LIN {X 7.026,Y 51.847,Z 52.000,A 180.000,B 0.000,C 180.000} C_DIS
LIN {X 6.520,Y 53.277,Z 52.000,A 180.000,B 0.000,C 180.000} C_DIS
LIN {X 6.460,Y 53.455,Z 52.000,A 180.000,B 0.000,C 180.000} C_DIS
LIN {X 5.992,Y 54.886,Z 52.000,A 180.000,B 0.000,C 180.000} C_DIS
LIN {X 5.935,Y 55.064,Z 52.000,A 180.000,B 0.000,C 180.000} C_DIS
LIN {X 5.503,Y 56.495,Z 52.000,A 180.000,B 0.000,C 180.000} C_DIS
LIN {X 5.450,Y 56.673,Z 52.000,A 180.000,B 0.000,C 180.000} C_DIS
LIN {X 5.400,Y 56.852,Z 52.000,A 180.000,B 0.000,C 180.000} C_DIS
LIN {X 5.005,Y 58.282,Z 52.000,A 180.000,B 0.000,C 180.000} C_DIS
LIN {X 4.958,Y 58.461,Z 52.000,A 180.000,B 0.000,C 180.000} C_DIS
LIN {X 4.598,Y 59.891,Z 52.000,A 180.000,B 0.000,C 180.000} C_DIS
LIN {X 4.554,Y 60.070,Z 52.000,A 180.000,B 0.000,C 180.000} C_DIS
LIN {X 4.513,Y 60.249,Z 52.000,A 180.000,B 0.000,C 180.000} C_DIS
LIN {X 4.189,Y 61.679,Z 52.000,A 180.000,B 0.000,C 180.000} C_DIS
LIN {X 4.150,Y 61.858,Z 52.000,A 180.000,B 0.000,C 180.000} C_DIS
LIN {X 3.825,Y 63.467,Z 52.000,A 180.000,B 0.000,C 180.000} C_DIS
LIN {X 3.792,Y 63.645,Z 52.000,A 180.000,B 0.000,C 180.000} C_DIS
LIN {X 3.538,Y 65.075,Z 52.000,A 180.000,B 0.000,C 180.000} C_DIS
LIN {X 3.506,Y 65.254,Z 52.000,A 180.000,B 0.000,C 180.000} C_DIS
LIN {X 3.479,Y 65.433,Z 52.000,A 180.000,B 0.000,C 180.000} C_DIS
LIN {X 3.259,Y 66.863,Z 52.000,A 180.000,B 0.000,C 180.000} C_DIS
LIN {X 3.233,Y 67.042,Z 52.000,A 180.000,B 0.000,C 180.000} C_DIS
LIN {X 3.025,Y 68.651,Z 52.000,A 180.000,B 0.000,C 180.000} C_DIS
LIN {X 3.004,Y 68.830,Z 52.000,A 180.000,B 0.000,C 180.000} C_DIS
LIN {X 2.833,Y 70.439,Z 52.000,A 180.000,B 0.000,C 180.000} C_DIS
LIN {X 2.818,Y 70.617,Z 52.000,A 180.000,B 0.000,C 180.000} C_DIS
LIN {X 2.700,Y 72.048,Z 52.000,A 180.000,B 0.000,C 180.000} C_DIS
LIN {X 2.686,Y 72.226,Z 52.000,A 180.000,B 0.000,C 180.000} C_DIS
LIN {X 2.685,Y 72.239,Z 52.000,A 180.000,B 0.000,C 180.000} C_DIS
LIN {X 2.675,Y 72.405,Z 52.000,A 180.000,B 0.000,C 180.000} C_DIS
LIN {X 2.591,Y 73.835,Z 52.000,A 180.000,B 0.000,C 180.000} C_DIS
LIN {X 2.581,Y 74.014,Z 52.000,A 180.000,B 0.000,C 180.000} C_DIS
LIN {X 2.525,Y 75.623,Z 52.000,A 180.000,B 0.000,C 180.000} C_DIS
LIN {X 2.520,Y 75.802,Z 52.000,A 180.000,B 0.000,C 180.000} C_DIS
LIN {X 2.506,Y 76.973,Z 52.000,A 180.000,B 0.000,C 180.000} C_DIS
LIN {X 2.501,Y 77.411,Z 52.000,A 180.000,B 0.000,C 180.000} C_DIS
LIN {X 2.501,Y 77.589,Z 52.000,A 180.000,B 0.000,C 180.000} C_DIS
LIN {X 2.520,Y 79.198,Z 52.000,A 180.000,B 0.000,C 180.000} C_DIS
LIN {X 2.525,Y 79.377,Z 52.000,A 180.000,B 0.000,C 180.000} C_DIS
LIN {X 2.581,Y 80.986,Z 52.000,A 180.000,B 0.000,C 180.000} C_DIS
LIN {X 2.591,Y 81.165,Z 52.000,A 180.000,B 0.000,C 180.000} C_DIS
LIN {X 2.675,Y 82.595,Z 52.000,A 180.000,B 0.000,C 180.000} C_DIS
LIN {X 2.685,Y 82.761,Z 52.000,A 180.000,B 0.000,C 180.000} C_DIS
LIN {X 2.686,Y 82.774,Z 52.000,A 180.000,B 0.000,C 180.000} C_DIS
LIN {X 2.700,Y 82.952,Z 52.000,A 180.000,B 0.000,C 180.000} C_DIS
LIN {X 2.818,Y 84.383,Z 52.000,A 180.000,B 0.000,C 180.000} C_DIS
LIN {X 2.833,Y 84.561,Z 52.000,A 180.000,B 0.000,C 180.000} C_DIS
LIN {X 3.004,Y 86.170,Z 52.000,A 180.000,B 0.000,C 180.000} C_DIS
LIN {X 3.025,Y 86.349,Z 52.000,A 180.000,B 0.000,C 180.000} C_DIS
LIN {X 3.233,Y 87.958,Z 52.000,A 180.000,B 0.000,C 180.000} C_DIS
LIN {X 3.259,Y 88.137,Z 52.000,A 180.000,B 0.000,C 180.000} C_DIS
LIN {X 3.479,Y 89.567,Z 52.000,A 180.000,B 0.000,C 180.000} C_DIS
LIN {X 3.506,Y 89.746,Z 52.000,A 180.000,B 0.000,C 180.000} C_DIS
LIN {X 3.538,Y 89.925,Z 52.000,A 180.000,B 0.000,C 180.000} C_DIS
LIN {X 3.792,Y 91.355,Z 52.000,A 180.000,B 0.000,C 180.000} C_DIS
LIN {X 3.825,Y 91.533,Z 52.000,A 180.000,B 0.000,C 180.000} C_DIS
LIN {X 4.150,Y 93.142,Z 52.000,A 180.000,B 0.000,C 180.000} C_DIS
LIN {X 4.189,Y 93.321,Z 52.000,A 180.000,B 0.000,C 180.000} C_DIS
LIN {X 4.513,Y 94.751,Z 52.000,A 180.000,B 0.000,C 180.000} C_DIS
LIN {X 4.554,Y 94.930,Z 52.000,A 180.000,B 0.000,C 180.000} C_DIS
LIN {X 4.598,Y 95.109,Z 52.000,A 180.000,B 0.000,C 180.000} C_DIS
LIN {X 4.958,Y 96.539,Z 52.000,A 180.000,B 0.000,C 180.000} C_DIS
LIN {X 5.005,Y 96.718,Z 52.000,A 180.000,B 0.000,C 180.000} C_DIS
LIN {X 5.400,Y 98.148,Z 52.000,A 180.000,B 0.000,C 180.000} C_DIS
LIN {X 5.450,Y 98.327,Z 52.000,A 180.000,B 0.000,C 180.000} C_DIS
LIN {X 5.503,Y 98.505,Z 52.000,A 180.000,B 0.000,C 180.000} C_DIS
LIN {X 5.935,Y 99.936,Z 52.000,A 180.000,B 0.000,C 180.000} C_DIS
LIN {X 5.992,Y 100.114,Z 52.000,A 180.000,B 0.000,C 180.000} C_DIS
LIN {X 6.460,Y 101.545,Z 52.000,A 180.000,B 0.000,C 180.000} C_DIS
LIN {X 6.520,Y 101.723,Z 52.000,A 180.000,B 0.000,C 180.000} C_DIS
LIN {X 7.026,Y 103.153,Z 52.000,A 180.000,B 0.000,C 180.000} C_DIS
LIN {X 7.089,Y 103.332,Z 52.000,A 180.000,B 0.000,C 180.000} C_DIS
LIN {X 7.154,Y 103.504,Z 52.000,A 180.000,B 0.000,C 180.000} C_DIS
LIN {X 7.701,Y 104.941,Z 52.000,A 180.000,B 0.000,C 180.000} C_DIS
LIN {X 7.773,Y 105.120,Z 52.000,A 180.000,B 0.000,C 180.000} C_DIS
LIN {X 8.355,Y 106.550,Z 52.000,A 180.000,B 0.000,C 180.000} C_DIS
LIN {X 8.405,Y 106.669,Z 52.000,A 180.000,B 0.000,C 180.000} C_DIS
LIN {X 9.053,Y 108.159,Z 52.000,A 180.000,B 0.000,C 180.000} C_DIS
LIN {X 9.120,Y 108.308,Z 52.000,A 180.000,B 0.000,C 180.000} C_DIS
LIN {X 9.797,Y 109.768,Z 52.000,A 180.000,B 0.000,C 180.000} C_DIS
LIN {X 9.836,Y 109.849,Z 52.000,A 180.000,B 0.000,C 180.000} C_DIS
LIN {X 10.551,Y 111.303,Z 52.000,A 180.000,B 0.000,C 180.000} C_DIS
LIN {X 10.587,Y 111.377,Z 52.000,A 180.000,B 0.000,C 180.000} C_DIS
LIN {X 10.680,Y 111.556,Z 52.000,A 180.000,B 0.000,C 180.000} C_DIS
LIN {X 11.332,Y 112.807,Z 52.000,A 180.000,B 0.000,C 180.000} C_DIS
LIN {X 11.426,Y 112.986,Z 52.000,A 180.000,B 0.000,C 180.000} C_DIS
LIN {X 12.215,Y 114.416,Z 52.000,A 180.000,B 0.000,C 180.000} C_DIS
LIN {X 12.317,Y 114.595,Z 52.000,A 180.000,B 0.000,C 180.000} C_DIS
LIN {X 13.053,Y 115.859,Z 52.000,A 180.000,B 0.000,C 180.000} C_DIS
LIN {X 13.151,Y 116.025,Z 52.000,A 180.000,B 0.000,C 180.000} C_DIS
LIN {X 13.232,Y 116.158,Z 52.000,A 180.000,B 0.000,C 180.000} C_DIS
LIN {X 14.029,Y 117.455,Z 52.000,A 180.000,B 0.000,C 180.000} C_DIS
LIN {X 14.126,Y 117.607,Z 52.000,A 180.000,B 0.000,C 180.000} C_DIS
LIN {X 14.953,Y 118.885,Z 52.000,A 180.000,B 0.000,C 180.000} C_DIS
LIN {X 15.020,Y 118.988,Z 52.000,A 180.000,B 0.000,C 180.000} C_DIS
LIN {X 15.072,Y 119.064,Z 52.000,A 180.000,B 0.000,C 180.000} C_DIS
LIN {X 15.924,Y 120.315,Z 52.000,A 180.000,B 0.000,C 180.000} C_DIS
LIN {X 16.047,Y 120.494,Z 52.000,A 180.000,B 0.000,C 180.000} C_DIS
LIN {X 16.986,Y 121.806,Z 52.000,A 180.000,B 0.000,C 180.000} C_DIS
LIN {X 17.073,Y 121.924,Z 52.000,A 180.000,B 0.000,C 180.000} C_DIS
LIN {X 18.059,Y 123.235,Z 52.000,A 180.000,B 0.000,C 180.000} C_DIS
LIN {X 18.152,Y 123.354,Z 52.000,A 180.000,B 0.000,C 180.000} C_DIS
LIN {X 19.139,Y 124.606,Z 52.000,A 180.000,B 0.000,C 180.000} C_DIS
LIN {X 19.286,Y 124.785,Z 52.000,A 180.000,B 0.000,C 180.000} C_DIS
LIN {X 20.204,Y 125.894,Z 52.000,A 180.000,B 0.000,C 180.000} C_DIS
LIN {X 20.323,Y 126.036,Z 52.000,A 180.000,B 0.000,C 180.000} C_DIS
LIN {X 21.410,Y 127.287,Z 52.000,A 180.000,B 0.000,C 180.000} C_DIS
LIN {X 21.456,Y 127.340,Z 52.000,A 180.000,B 0.000,C 180.000} C_DIS
LIN {X 21.570,Y 127.466,Z 52.000,A 180.000,B 0.000,C 180.000} C_DIS
LIN {X 22.547,Y 128.539,Z 52.000,A 180.000,B 0.000,C 180.000} C_DIS
LIN {X 22.707,Y 128.711,Z 52.000,A 180.000,B 0.000,C 180.000} C_DIS
LIN {X 23.780,Y 129.835,Z 52.000,A 180.000,B 0.000,C 180.000} C_DIS
LIN {X 23.910,Y 129.969,Z 52.000,A 180.000,B 0.000,C 180.000} C_DIS
LIN {X 25.031,Y 131.090,Z 52.000,A 180.000,B 0.000,C 180.000} C_DIS
LIN {X 25.165,Y 131.220,Z 52.000,A 180.000,B 0.000,C 180.000} C_DIS
LIN {X 26.289,Y 132.293,Z 52.000,A 180.000,B 0.000,C 180.000} C_DIS
LIN {X 26.461,Y 132.453,Z 52.000,A 180.000,B 0.000,C 180.000} C_DIS
LIN {X 27.534,Y 133.430,Z 52.000,A 180.000,B 0.000,C 180.000} C_DIS
LIN {X 27.660,Y 133.544,Z 52.000,A 180.000,B 0.000,C 180.000} C_DIS
LIN {X 27.713,Y 133.590,Z 52.000,A 180.000,B 0.000,C 180.000} C_DIS
LIN {X 28.964,Y 134.677,Z 52.000,A 180.000,B 0.000,C 180.000} C_DIS
LIN {X 29.106,Y 134.796,Z 52.000,A 180.000,B 0.000,C 180.000} C_DIS
LIN {X 30.215,Y 135.714,Z 52.000,A 180.000,B 0.000,C 180.000} C_DIS
LIN {X 30.394,Y 135.861,Z 52.000,A 180.000,B 0.000,C 180.000} C_DIS
LIN {X 31.646,Y 136.848,Z 52.000,A 180.000,B 0.000,C 180.000} C_DIS
LIN {X 31.765,Y 136.941,Z 52.000,A 180.000,B 0.000,C 180.000} C_DIS
LIN {X 33.076,Y 137.927,Z 52.000,A 180.000,B 0.000,C 180.000} C_DIS
LIN {X 33.194,Y 138.014,Z 52.000,A 180.000,B 0.000,C 180.000} C_DIS
LIN {X 34.506,Y 138.953,Z 52.000,A 180.000,B 0.000,C 180.000} C_DIS
LIN {X 34.685,Y 139.076,Z 52.000,A 180.000,B 0.000,C 180.000} C_DIS
LIN {X 35.936,Y 139.928,Z 52.000,A 180.000,B 0.000,C 180.000} C_DIS
LIN {X 36.012,Y 139.980,Z 52.000,A 180.000,B 0.000,C 180.000} C_DIS
LIN {X 36.115,Y 140.047,Z 52.000,A 180.000,B 0.000,C 180.000} C_DIS
LIN {X 37.393,Y 140.874,Z 52.000,A 180.000,B 0.000,C 180.000} C_DIS
LIN {X 37.545,Y 140.971,Z 52.000,A 180.000,B 0.000,C 180.000} C_DIS
LIN {X 38.842,Y 141.768,Z 52.000,A 180.000,B 0.000,C 180.000} C_DIS
LIN {X 38.975,Y 141.849,Z 52.000,A 180.000,B 0.000,C 180.000} C_DIS
LIN {X 39.141,Y 141.947,Z 52.000,A 180.000,B 0.000,C 180.000} C_DIS
LIN {X 40.405,Y 142.683,Z 52.000,A 180.000,B 0.000,C 180.000} C_DIS
LIN {X 40.584,Y 142.785,Z 52.000,A 180.000,B 0.000,C 180.000} C_DIS
LIN {X 42.014,Y 143.574,Z 52.000,A 180.000,B 0.000,C 180.000} C_DIS
LIN {X 42.193,Y 143.668,Z 52.000,A 180.000,B 0.000,C 180.000} C_DIS
LIN {X 43.444,Y 144.320,Z 52.000,A 180.000,B 0.000,C 180.000} C_DIS
LIN {X 43.623,Y 144.413,Z 52.000,A 180.000,B 0.000,C 180.000} C_DIS
LIN {X 43.697,Y 144.449,Z 52.000,A 180.000,B 0.000,C 180.000} C_DIS
LIN {X 45.151,Y 145.164,Z 52.000,A 180.000,B 0.000,C 180.000} C_DIS
LIN {X 45.232,Y 145.203,Z 52.000,A 180.000,B 0.000,C 180.000} C_DIS
LIN {X 46.692,Y 145.880,Z 52.000,A 180.000,B 0.000,C 180.000} C_DIS
LIN {X 46.841,Y 145.947,Z 52.000,A 180.000,B 0.000,C 180.000} C_DIS
LIN {X 48.331,Y 146.595,Z 52.000,A 180.000,B 0.000,C 180.000} C_DIS
LIN {X 48.450,Y 146.645,Z 52.000,A 180.000,B 0.000,C 180.000} C_DIS
LIN {X 49.880,Y 147.227,Z 52.000,A 180.000,B 0.000,C 180.000} C_DIS
LIN {X 50.059,Y 147.299,Z 52.000,A 180.000,B 0.000,C 180.000} C_DIS
LIN {X 51.496,Y 147.846,Z 52.000,A 180.000,B 0.000,C 180.000} C_DIS
LIN {X 51.668,Y 147.911,Z 52.000,A 180.000,B 0.000,C 180.000} C_DIS
LIN {X 51.847,Y 147.974,Z 52.000,A 180.000,B 0.000,C 180.000} C_DIS
LIN {X 53.277,Y 148.480,Z 52.000,A 180.000,B 0.000,C 180.000} C_DIS
LIN {X 53.455,Y 148.540,Z 52.000,A 180.000,B 0.000,C 180.000} C_DIS
LIN {X 54.290,Y 148.813,Z 52.000,A 180.000,B 0.000,C 180.000} C_DIS
LIN {X 54.886,Y 149.008,Z 52.000,A 180.000,B 0.000,C 180.000} C_DIS
LIN {X 55.064,Y 149.065,Z 52.000,A 180.000,B 0.000,C 180.000} C_DIS
LIN {X 56.495,Y 149.497,Z 52.000,A 180.000,B 0.000,C 180.000} C_DIS
LIN {X 56.673,Y 149.550,Z 52.000,A 180.000,B 0.000,C 180.000} C_DIS
LIN {X 56.852,Y 149.600,Z 52.000,A 180.000,B 0.000,C 180.000} C_DIS
LIN {X 58.282,Y 149.995,Z 52.000,A 180.000,B 0.000,C 180.000} C_DIS
LIN {X 58.461,Y 150.042,Z 52.000,A 180.000,B 0.000,C 180.000} C_DIS
LIN {X 59.891,Y 150.402,Z 52.000,A 180.000,B 0.000,C 180.000} C_DIS
LIN {X 60.070,Y 150.447,Z 52.000,A 180.000,B 0.000,C 180.000} C_DIS
LIN {X 60.249,Y 150.487,Z 52.000,A 180.000,B 0.000,C 180.000} C_DIS
LIN {X 61.679,Y 150.811,Z 52.000,A 180.000,B 0.000,C 180.000} C_DIS
LIN {X 61.858,Y 150.850,Z 52.000,A 180.000,B 0.000,C 180.000} C_DIS
LIN {X 63.467,Y 151.175,Z 52.000,A 180.000,B 0.000,C 180.000} C_DIS
LIN {X 63.645,Y 151.208,Z 52.000,A 180.000,B 0.000,C 180.000} C_DIS
LIN {X 65.075,Y 151.462,Z 52.000,A 180.000,B 0.000,C 180.000} C_DIS
LIN {X 65.254,Y 151.494,Z 52.000,A 180.000,B 0.000,C 180.000} C_DIS
LIN {X 65.433,Y 151.521,Z 52.000,A 180.000,B 0.000,C 180.000} C_DIS
LIN {X 66.863,Y 151.741,Z 52.000,A 180.000,B 0.000,C 180.000} C_DIS
LIN {X 67.042,Y 151.767,Z 52.000,A 180.000,B 0.000,C 180.000} C_DIS
LIN {X 68.651,Y 151.975,Z 52.000,A 180.000,B 0.000,C 180.000} C_DIS
LIN {X 68.830,Y 151.996,Z 52.000,A 180.000,B 0.000,C 180.000} C_DIS
LIN {X 70.439,Y 152.167,Z 52.000,A 180.000,B 0.000,C 180.000} C_DIS
LIN {X 70.617,Y 152.182,Z 52.000,A 180.000,B 0.000,C 180.000} C_DIS
LIN {X 72.048,Y 152.300,Z 52.000,A 180.000,B 0.000,C 180.000} C_DIS
LIN {X 72.226,Y 152.314,Z 52.000,A 180.000,B 0.000,C 180.000} C_DIS
LIN {X 72.239,Y 152.315,Z 52.000,A 180.000,B 0.000,C 180.000} C_DIS
LIN {X 72.405,Y 152.325,Z 52.000,A 180.000,B 0.000,C 180.000} C_DIS
LIN {X 73.835,Y 152.409,Z 52.000,A 180.000,B 0.000,C 180.000} C_DIS
LIN {X 74.014,Y 152.419,Z 52.000,A 180.000,B 0.000,C 180.000} C_DIS
LIN {X 75.623,Y 152.475,Z 52.000,A 180.000,B 0.000,C 180.000} C_DIS
LIN {X 75.802,Y 152.480,Z 52.000,A 180.000,B 0.000,C 180.000} C_DIS
LIN {X 77.411,Y 152.499,Z 52.000,A 180.000,B 0.000,C 180.000} C_DIS
LIN {X 77.589,Y 152.499,Z 52.000,A 180.000,B 0.000,C 180.000} C_DIS
LIN {X 79.198,Y 152.480,Z 52.000,A 180.000,B 0.000,C 180.000} C_DIS
LIN {X 79.377,Y 152.475,Z 52.000,A 180.000,B 0.000,C 180.000} C_DIS
LIN {X 80.986,Y 152.419,Z 52.000,A 180.000,B 0.000,C 180.000} C_DIS
LIN {X 81.165,Y 152.409,Z 52.000,A 180.000,B 0.000,C 180.000} C_DIS
LIN {X 82.595,Y 152.325,Z 52.000,A 180.000,B 0.000,C 180.000} C_DIS
LIN {X 82.761,Y 152.315,Z 52.000,A 180.000,B 0.000,C 180.000} C_DIS
LIN {X 82.774,Y 152.314,Z 52.000,A 180.000,B 0.000,C 180.000} C_DIS
LIN {X 82.952,Y 152.300,Z 52.000,A 180.000,B 0.000,C 180.000} C_DIS
LIN {X 84.383,Y 152.182,Z 52.000,A 180.000,B 0.000,C 180.000} C_DIS
LIN {X 84.561,Y 152.167,Z 52.000,A 180.000,B 0.000,C 180.000} C_DIS
LIN {X 86.170,Y 151.996,Z 52.000,A 180.000,B 0.000,C 180.000} C_DIS
LIN {X 86.349,Y 151.975,Z 52.000,A 180.000,B 0.000,C 180.000} C_DIS
LIN {X 87.958,Y 151.767,Z 52.000,A 180.000,B 0.000,C 180.000} C_DIS
LIN {X 88.137,Y 151.741,Z 52.000,A 180.000,B 0.000,C 180.000} C_DIS
LIN {X 89.567,Y 151.521,Z 52.000,A 180.000,B 0.000,C 180.000} C_DIS
LIN {X 89.746,Y 151.494,Z 52.000,A 180.000,B 0.000,C 180.000} C_DIS
LIN {X 89.925,Y 151.462,Z 52.000,A 180.000,B 0.000,C 180.000} C_DIS
LIN {X 91.355,Y 151.208,Z 52.000,A 180.000,B 0.000,C 180.000} C_DIS
LIN {X 91.533,Y 151.175,Z 52.000,A 180.000,B 0.000,C 180.000} C_DIS
LIN {X 93.142,Y 150.850,Z 52.000,A 180.000,B 0.000,C 180.000} C_DIS
LIN {X 93.321,Y 150.811,Z 52.000,A 180.000,B 0.000,C 180.000} C_DIS
LIN {X 94.751,Y 150.487,Z 52.000,A 180.000,B 0.000,C 180.000} C_DIS
LIN {X 94.930,Y 150.447,Z 52.000,A 180.000,B 0.000,C 180.000} C_DIS
LIN {X 95.109,Y 150.402,Z 52.000,A 180.000,B 0.000,C 180.000} C_DIS
LIN {X 96.539,Y 150.042,Z 52.000,A 180.000,B 0.000,C 180.000} C_DIS
LIN {X 96.718,Y 149.995,Z 52.000,A 180.000,B 0.000,C 180.000} C_DIS
LIN {X 98.148,Y 149.600,Z 52.000,A 180.000,B 0.000,C 180.000} C_DIS
LIN {X 98.327,Y 149.550,Z 52.000,A 180.000,B 0.000,C 180.000} C_DIS
LIN {X 98.505,Y 149.497,Z 52.000,A 180.000,B 0.000,C 180.000} C_DIS
LIN {X 99.936,Y 149.065,Z 52.000,A 180.000,B 0.000,C 180.000} C_DIS
LIN {X 100.114,Y 149.008,Z 52.000,A 180.000,B 0.000,C 180.000} C_DIS
LIN {X 101.545,Y 148.540,Z 52.000,A 180.000,B 0.000,C 180.000} C_DIS
LIN {X 101.723,Y 148.480,Z 52.000,A 180.000,B 0.000,C 180.000} C_DIS
LIN {X 103.153,Y 147.974,Z 52.000,A 180.000,B 0.000,C 180.000} C_DIS
LIN {X 103.332,Y 147.911,Z 52.000,A 180.000,B 0.000,C 180.000} C_DIS
LIN {X 103.504,Y 147.846,Z 52.000,A 180.000,B 0.000,C 180.000} C_DIS
LIN {X 104.941,Y 147.299,Z 52.000,A 180.000,B 0.000,C 180.000} C_DIS
LIN {X 105.120,Y 147.227,Z 52.000,A 180.000,B 0.000,C 180.000} C_DIS
LIN {X 106.550,Y 146.645,Z 52.000,A 180.000,B 0.000,C 180.000} C_DIS
LIN {X 106.669,Y 146.595,Z 52.000,A 180.000,B 0.000,C 180.000} C_DIS
LIN {X 108.159,Y 145.947,Z 52.000,A 180.000,B 0.000,C 180.000} C_DIS
LIN {X 108.308,Y 145.880,Z 52.000,A 180.000,B 0.000,C 180.000} C_DIS
LIN {X 109.768,Y 145.203,Z 52.000,A 180.000,B 0.000,C 180.000} C_DIS
LIN {X 109.849,Y 145.164,Z 52.000,A 180.000,B 0.000,C 180.000} C_DIS
LIN {X 111.303,Y 144.449,Z 52.000,A 180.000,B 0.000,C 180.000} C_DIS
LIN {X 111.377,Y 144.413,Z 52.000,A 180.000,B 0.000,C 180.000} C_DIS
LIN {X 111.556,Y 144.320,Z 52.000,A 180.000,B 0.000,C 180.000} C_DIS
LIN {X 112.807,Y 143.668,Z 52.000,A 180.000,B 0.000,C 180.000} C_DIS
LIN {X 112.986,Y 143.574,Z 52.000,A 180.000,B 0.000,C 180.000} C_DIS
LIN {X 114.416,Y 142.785,Z 52.000,A 180.000,B 0.000,C 180.000} C_DIS
LIN {X 114.595,Y 142.683,Z 52.000,A 180.000,B 0.000,C 180.000} C_DIS
LIN {X 115.859,Y 141.947,Z 52.000,A 180.000,B 0.000,C 180.000} C_DIS
LIN {X 116.025,Y 141.849,Z 52.000,A 180.000,B 0.000,C 180.000} C_DIS
LIN {X 116.158,Y 141.768,Z 52.000,A 180.000,B 0.000,C 180.000} C_DIS
LIN {X 117.455,Y 140.971,Z 52.000,A 180.000,B 0.000,C 180.000} C_DIS
LIN {X 117.607,Y 140.874,Z 52.000,A 180.000,B 0.000,C 180.000} C_DIS
LIN {X 118.885,Y 140.047,Z 52.000,A 180.000,B 0.000,C 180.000} C_DIS
LIN {X 118.988,Y 139.980,Z 52.000,A 180.000,B 0.000,C 180.000} C_DIS
LIN {X 119.064,Y 139.928,Z 52.000,A 180.000,B 0.000,C 180.000} C_DIS
LIN {X 120.315,Y 139.076,Z 52.000,A 180.000,B 0.000,C 180.000} C_DIS
LIN {X 120.494,Y 138.953,Z 52.000,A 180.000,B 0.000,C 180.000} C_DIS
LIN {X 121.806,Y 138.014,Z 52.000,A 180.000,B 0.000,C 180.000} C_DIS
LIN {X 121.924,Y 137.927,Z 52.000,A 180.000,B 0.000,C 180.000} C_DIS
LIN {X 123.235,Y 136.941,Z 52.000,A 180.000,B 0.000,C 180.000} C_DIS
LIN {X 123.354,Y 136.848,Z 52.000,A 180.000,B 0.000,C 180.000} C_DIS
LIN {X 124.606,Y 135.861,Z 52.000,A 180.000,B 0.000,C 180.000} C_DIS
LIN {X 124.785,Y 135.714,Z 52.000,A 180.000,B 0.000,C 180.000} C_DIS
LIN {X 125.894,Y 134.796,Z 52.000,A 180.000,B 0.000,C 180.000} C_DIS
LIN {X 126.036,Y 134.677,Z 52.000,A 180.000,B 0.000,C 180.000} C_DIS
LIN {X 127.287,Y 133.590,Z 52.000,A 180.000,B 0.000,C 180.000} C_DIS
LIN {X 127.340,Y 133.544,Z 52.000,A 180.000,B 0.000,C 180.000} C_DIS
LIN {X 127.466,Y 133.430,Z 52.000,A 180.000,B 0.000,C 180.000} C_DIS
LIN {X 128.539,Y 132.453,Z 52.000,A 180.000,B 0.000,C 180.000} C_DIS
LIN {X 128.711,Y 132.293,Z 52.000,A 180.000,B 0.000,C 180.000} C_DIS
LIN {X 129.835,Y 131.220,Z 52.000,A 180.000,B 0.000,C 180.000} C_DIS
LIN {X 129.969,Y 131.090,Z 52.000,A 180.000,B 0.000,C 180.000} C_DIS
LIN {X 131.090,Y 129.969,Z 52.000,A 180.000,B 0.000,C 180.000} C_DIS
LIN {X 131.220,Y 129.835,Z 52.000,A 180.000,B 0.000,C 180.000} C_DIS
LIN {X 132.293,Y 128.711,Z 52.000,A 180.000,B 0.000,C 180.000} C_DIS
LIN {X 132.453,Y 128.539,Z 52.000,A 180.000,B 0.000,C 180.000} C_DIS
LIN {X 133.430,Y 127.466,Z 52.000,A 180.000,B 0.000,C 180.000} C_DIS
LIN {X 133.544,Y 127.340,Z 52.000,A 180.000,B 0.000,C 180.000} C_DIS
LIN {X 133.590,Y 127.287,Z 52.000,A 180.000,B 0.000,C 180.000} C_DIS
LIN {X 134.677,Y 126.036,Z 52.000,A 180.000,B 0.000,C 180.000} C_DIS
LIN {X 134.796,Y 125.894,Z 52.000,A 180.000,B 0.000,C 180.000} C_DIS
LIN {X 135.714,Y 124.785,Z 52.000,A 180.000,B 0.000,C 180.000} C_DIS
LIN {X 135.861,Y 124.606,Z 52.000,A 180.000,B 0.000,C 180.000} C_DIS
LIN {X 136.848,Y 123.354,Z 52.000,A 180.000,B 0.000,C 180.000} C_DIS
LIN {X 136.941,Y 123.235,Z 52.000,A 180.000,B 0.000,C 180.000} C_DIS
LIN {X 137.927,Y 121.924,Z 52.000,A 180.000,B 0.000,C 180.000} C_DIS
LIN {X 138.014,Y 121.806,Z 52.000,A 180.000,B 0.000,C 180.000} C_DIS
LIN {X 138.953,Y 120.494,Z 52.000,A 180.000,B 0.000,C 180.000} C_DIS
LIN {X 139.076,Y 120.315,Z 52.000,A 180.000,B 0.000,C 180.000} C_DIS
LIN {X 139.928,Y 119.064,Z 52.000,A 180.000,B 0.000,C 180.000} C_DIS
LIN {X 139.980,Y 118.988,Z 52.000,A 180.000,B 0.000,C 180.000} C_DIS
LIN {X 140.047,Y 118.885,Z 52.000,A 180.000,B 0.000,C 180.000} C_DIS
LIN {X 140.874,Y 117.607,Z 52.000,A 180.000,B 0.000,C 180.000} C_DIS
LIN {X 140.971,Y 117.455,Z 52.000,A 180.000,B 0.000,C 180.000} C_DIS
LIN {X 141.768,Y 116.158,Z 52.000,A 180.000,B 0.000,C 180.000} C_DIS
LIN {X 141.849,Y 116.025,Z 52.000,A 180.000,B 0.000,C 180.000} C_DIS
LIN {X 141.947,Y 115.859,Z 52.000,A 180.000,B 0.000,C 180.000} C_DIS
LIN {X 142.683,Y 114.595,Z 52.000,A 180.000,B 0.000,C 180.000} C_DIS
LIN {X 142.785,Y 114.416,Z 52.000,A 180.000,B 0.000,C 180.000} C_DIS
LIN {X 143.574,Y 112.986,Z 52.000,A 180.000,B 0.000,C 180.000} C_DIS
LIN {X 143.668,Y 112.807,Z 52.000,A 180.000,B 0.000,C 180.000} C_DIS
LIN {X 144.320,Y 111.556,Z 52.000,A 180.000,B 0.000,C 180.000} C_DIS
LIN {X 144.413,Y 111.377,Z 52.000,A 180.000,B 0.000,C 180.000} C_DIS
LIN {X 144.449,Y 111.303,Z 52.000,A 180.000,B 0.000,C 180.000} C_DIS
LIN {X 145.164,Y 109.849,Z 52.000,A 180.000,B 0.000,C 180.000} C_DIS
LIN {X 145.203,Y 109.768,Z 52.000,A 180.000,B 0.000,C 180.000} C_DIS
LIN {X 145.656,Y 108.791,Z 52.000,A 180.000,B 0.000,C 180.000} C_DIS
LIN {X 145.880,Y 108.308,Z 52.000,A 180.000,B 0.000,C 180.000} C_DIS
LIN {X 145.947,Y 108.159,Z 52.000,A 180.000,B 0.000,C 180.000} C_DIS
LIN {X 146.595,Y 106.669,Z 52.000,A 180.000,B 0.000,C 180.000} C_DIS
LIN {X 146.645,Y 106.550,Z 52.000,A 180.000,B 0.000,C 180.000} C_DIS
LIN {X 147.227,Y 105.120,Z 52.000,A 180.000,B 0.000,C 180.000} C_DIS
LIN {X 147.299,Y 104.941,Z 52.000,A 180.000,B 0.000,C 180.000} C_DIS
LIN {X 147.846,Y 103.504,Z 52.000,A 180.000,B 0.000,C 180.000} C_DIS
LIN {X 147.911,Y 103.332,Z 52.000,A 180.000,B 0.000,C 180.000} C_DIS
LIN {X 147.974,Y 103.153,Z 52.000,A 180.000,B 0.000,C 180.000} C_DIS
LIN {X 148.480,Y 101.723,Z 52.000,A 180.000,B 0.000,C 180.000} C_DIS
LIN {X 148.540,Y 101.545,Z 52.000,A 180.000,B 0.000,C 180.000} C_DIS
LIN {X 149.008,Y 100.114,Z 52.000,A 180.000,B 0.000,C 180.000} C_DIS
LIN {X 149.065,Y 99.936,Z 52.000,A 180.000,B 0.000,C 180.000} C_DIS
LIN {X 149.497,Y 98.505,Z 52.000,A 180.000,B 0.000,C 180.000} C_DIS
LIN {X 149.550,Y 98.327,Z 52.000,A 180.000,B 0.000,C 180.000} C_DIS
LIN {X 149.600,Y 98.148,Z 52.000,A 180.000,B 0.000,C 180.000} C_DIS
LIN {X 149.995,Y 96.718,Z 52.000,A 180.000,B 0.000,C 180.000} C_DIS
LIN {X 150.042,Y 96.539,Z 52.000,A 180.000,B 0.000,C 180.000} C_DIS
LIN {X 150.402,Y 95.109,Z 52.000,A 180.000,B 0.000,C 180.000} C_DIS
LIN {X 150.447,Y 94.930,Z 52.000,A 180.000,B 0.000,C 180.000} C_DIS
LIN {X 150.487,Y 94.751,Z 52.000,A 180.000,B 0.000,C 180.000} C_DIS
LIN {X 150.811,Y 93.321,Z 52.000,A 180.000,B 0.000,C 180.000} C_DIS
LIN {X 150.850,Y 93.142,Z 52.000,A 180.000,B 0.000,C 180.000} C_DIS
LIN {X 151.175,Y 91.533,Z 52.000,A 180.000,B 0.000,C 180.000} C_DIS
LIN {X 151.208,Y 91.355,Z 52.000,A 180.000,B 0.000,C 180.000} C_DIS
LIN {X 151.462,Y 89.925,Z 52.000,A 180.000,B 0.000,C 180.000} C_DIS
LIN {X 151.494,Y 89.746,Z 52.000,A 180.000,B 0.000,C 180.000} C_DIS
LIN {X 151.521,Y 89.567,Z 52.000,A 180.000,B 0.000,C 180.000} C_DIS
LIN {X 151.741,Y 88.137,Z 52.000,A 180.000,B 0.000,C 180.000} C_DIS
LIN {X 151.767,Y 87.958,Z 52.000,A 180.000,B 0.000,C 180.000} C_DIS
LIN {X 151.975,Y 86.349,Z 52.000,A 180.000,B 0.000,C 180.000} C_DIS
LIN {X 151.996,Y 86.170,Z 52.000,A 180.000,B 0.000,C 180.000} C_DIS
LIN {X 152.167,Y 84.561,Z 52.000,A 180.000,B 0.000,C 180.000} C_DIS
LIN {X 152.182,Y 84.383,Z 52.000,A 180.000,B 0.000,C 180.000} C_DIS
LIN {X 152.300,Y 82.952,Z 52.000,A 180.000,B 0.000,C 180.000} C_DIS
LIN {X 152.314,Y 82.774,Z 52.000,A 180.000,B 0.000,C 180.000} C_DIS
LIN {X 152.315,Y 82.761,Z 52.000,A 180.000,B 0.000,C 180.000} C_DIS
LIN {X 152.325,Y 82.595,Z 52.000,A 180.000,B 0.000,C 180.000} C_DIS
LIN {X 152.409,Y 81.165,Z 52.000,A 180.000,B 0.000,C 180.000} C_DIS
LIN {X 152.419,Y 80.986,Z 52.000,A 180.000,B 0.000,C 180.000} C_DIS
LIN {X 152.475,Y 79.377,Z 52.000,A 180.000,B 0.000,C 180.000} C_DIS
LIN {X 152.480,Y 79.198,Z 52.000,A 180.000,B 0.000,C 180.000} C_DIS
LIN {X 152.499,Y 77.589,Z 52.000,A 180.000,B 0.000,C 180.000} C_DIS
LIN {X 152.499,Y 77.411,Z 52.000,A 180.000,B 0.000,C 180.000} C_DIS
LIN {X 152.480,Y 75.802,Z 52.000,A 180.000,B 0.000,C 180.000} C_DIS
LIN {X 152.475,Y 75.623,Z 52.000,A 180.000,B 0.000,C 180.000} C_DIS
LIN {X 152.419,Y 74.014,Z 52.000,A 180.000,B 0.000,C 180.000} C_DIS
LIN {X 152.409,Y 73.835,Z 52.000,A 180.000,B 0.000,C 180.000} C_DIS
LIN {X 152.342,Y 72.697,Z 52.000,A 180.000,B 0.000,C 180.000} C_DIS
; Lead Out Move Starts
LIN {X 152.468,Y 72.336,Z 52.000,A 180.000,B 0.000,C 180.000} C_DIS
LIN {X 152.812,Y 72.169,Z 52.000,A 180.000,B 0.000,C 180.000} C_DIS
; Link Move Starts
LIN {X 153.185,Y 71.967,Z 52.000,A 180.000,B 0.000,C 180.000} C_DIS
LIN {X 153.269,Y 71.551,Z 52.000,A 180.000,B 0.000,C 180.000} C_DIS
LIN {X 153.386,Y 71.095,Z 52.000,A 180.000,B 0.000,C 180.000} C_DIS
LIN {X 154.503,Y 70.413,Z 52.000,A 180.000,B 0.000,C 180.000} C_DIS
LIN {X 155.812,Y 70.426,Z 52.000,A 180.000,B 0.000,C 180.000} C_DIS
LIN {X 156.915,Y 71.130,Z 52.000,A 180.000,B 0.000,C 180.000} C_DIS
LIN {X 157.478,Y 72.311,Z 52.000,A 180.000,B 0.000,C 180.000} C_DIS
LIN {X 157.329,Y 73.611,Z 52.000,A 180.000,B 0.000,C 180.000} C_DIS
LIN {X 156.514,Y 74.635,Z 52.000,A 180.000,B 0.000,C 180.000} C_DIS
LIN {X 155.281,Y 75.073,Z 52.000,A 180.000,B 0.000,C 180.000} C_DIS
LIN {X 154.003,Y 74.790,Z 52.000,A 180.000,B 0.000,C 180.000} C_DIS
$VEL.CP=0.01
LIN {X 153.988,Y 74.782,Z 52.000,A 180.000,B 0.000,C 180.000} C_DIS
LIN {X 153.042,Y 73.825,Z 51.952,A 180.000,B 0.000,C 180.000} C_DIS
LIN {X 152.768,Y 72.509,Z 51.905,A 180.000,B 0.000,C 180.000} C_DIS
LIN {X 153.252,Y 71.255,Z 51.857,A 180.000,B 0.000,C 180.000} C_DIS
LIN {X 154.340,Y 70.464,Z 51.809,A 180.000,B 0.000,C 180.000} C_DIS
LIN {X 155.683,Y 70.391,Z 51.762,A 180.000,B 0.000,C 180.000} C_DIS
LIN {X 156.850,Y 71.059,Z 51.714,A 180.000,B 0.000,C 180.000} C_DIS
LIN {X 157.467,Y 72.254,Z 51.667,A 180.000,B 0.000,C 180.000} C_DIS
LIN {X 157.337,Y 73.592,Z 51.619,A 180.000,B 0.000,C 180.000} C_DIS
LIN {X 156.501,Y 74.645,Z 51.571,A 180.000,B 0.000,C 180.000} C_DIS
LIN {X 155.227,Y 75.075,Z 51.524,A 180.000,B 0.000,C 180.000} C_DIS
LIN {X 153.923,Y 74.745,Z 51.476,A 180.000,B 0.000,C 180.000} C_DIS
LIN {X 153.008,Y 73.759,Z 51.429,A 180.000,B 0.000,C 180.000} C_DIS
LIN {X 152.775,Y 72.435,Z 51.381,A 180.000,B 0.000,C 180.000} C_DIS
LIN {X 153.298,Y 71.196,Z 51.333,A 180.000,B 0.000,C 180.000} C_DIS
LIN {X 154.410,Y 70.440,Z 51.286,A 180.000,B 0.000,C 180.000} C_DIS
LIN {X 155.755,Y 70.409,Z 51.238,A 180.000,B 0.000,C 180.000} C_DIS
LIN {X 156.900,Y 71.114,Z 51.191,A 180.000,B 0.000,C 180.000} C_DIS
LIN {X 157.480,Y 72.327,Z 51.143,A 180.000,B 0.000,C 180.000} C_DIS
LIN {X 157.308,Y 73.661,Z 51.095,A 180.000,B 0.000,C 180.000} C_DIS
LIN {X 156.439,Y 74.687,Z 51.048,A 180.000,B 0.000,C 180.000} C_DIS
LIN {X 155.152,Y 75.077,Z 51.000,A 180.000,B 0.000,C 180.000} C_DIS
LIN {X 155.135,Y 75.077,Z 51.000,A 180.000,B 0.000,C 180.000} C_DIS
; Lead In Move Starts
LIN {X 154.880,Y 75.077,Z 51.000,A 180.000,B 0.000,C 180.000} C_DIS
LIN {X 153.690,Y 74.758,Z 51.000,A 180.000,B 0.000,C 180.000} C_DIS
LIN {X 152.819,Y 73.887,Z 51.000,A 180.000,B 0.000,C 180.000} C_DIS
LIN {X 152.500,Y 72.697,Z 51.000,A 180.000,B 0.000,C 180.000} C_DIS
; Cutting Move Starts
$VEL.CP=0.02
LIN {X 152.500,Y 5.009,Z 51.000,A 180.000,B 0.000,C 180.000} C_DIS
LIN {X 152.494,Y 4.830,Z 51.000,A 180.000,B 0.000,C 180.000} C_DIS
LIN {X 152.494,Y 4.827,Z 51.000,A 180.000,B 0.000,C 180.000} C_DIS
LIN {X 152.476,Y 4.651,Z 51.000,A 180.000,B 0.000,C 180.000} C_DIS
LIN {X 152.444,Y 4.472,Z 51.000,A 180.000,B 0.000,C 180.000} C_DIS
LIN {X 152.398,Y 4.294,Z 51.000,A 180.000,B 0.000,C 180.000} C_DIS
LIN {X 152.338,Y 4.115,Z 51.000,A 180.000,B 0.000,C 180.000} C_DIS
LIN {X 152.315,Y 4.057,Z 51.000,A 180.000,B 0.000,C 180.000} C_DIS
LIN {X 152.262,Y 3.936,Z 51.000,A 180.000,B 0.000,C 180.000} C_DIS
LIN {X 152.169,Y 3.757,Z 51.000,A 180.000,B 0.000,C 180.000} C_DIS
LIN {X 152.136,Y 3.702,Z 51.000,A 180.000,B 0.000,C 180.000} C_DIS
LIN {X 152.057,Y 3.579,Z 51.000,A 180.000,B 0.000,C 180.000} C_DIS
LIN {X 151.958,Y 3.445,Z 51.000,A 180.000,B 0.000,C 180.000} C_DIS
LIN {X 151.921,Y 3.400,Z 51.000,A 180.000,B 0.000,C 180.000} C_DIS
LIN {X 151.779,Y 3.243,Z 51.000,A 180.000,B 0.000,C 180.000} C_DIS
LIN {X 151.757,Y 3.221,Z 51.000,A 180.000,B 0.000,C 180.000} C_DIS
LIN {X 151.600,Y 3.079,Z 51.000,A 180.000,B 0.000,C 180.000} C_DIS
LIN {X 151.555,Y 3.042,Z 51.000,A 180.000,B 0.000,C 180.000} C_DIS
LIN {X 151.421,Y 2.943,Z 51.000,A 180.000,B 0.000,C 180.000} C_DIS
LIN {X 151.298,Y 2.864,Z 51.000,A 180.000,B 0.000,C 180.000} C_DIS
LIN {X 151.243,Y 2.831,Z 51.000,A 180.000,B 0.000,C 180.000} C_DIS
LIN {X 151.064,Y 2.738,Z 51.000,A 180.000,B 0.000,C 180.000} C_DIS
LIN {X 150.943,Y 2.685,Z 51.000,A 180.000,B 0.000,C 180.000} C_DIS
LIN {X 150.885,Y 2.662,Z 51.000,A 180.000,B 0.000,C 180.000} C_DIS
LIN {X 150.706,Y 2.602,Z 51.000,A 180.000,B 0.000,C 180.000} C_DIS
LIN {X 150.528,Y 2.556,Z 51.000,A 180.000,B 0.000,C 180.000} C_DIS
LIN {X 150.349,Y 2.524,Z 51.000,A 180.000,B 0.000,C 180.000} C_DIS
LIN {X 150.173,Y 2.506,Z 51.000,A 180.000,B 0.000,C 180.000} C_DIS
LIN {X 150.170,Y 2.506,Z 51.000,A 180.000,B 0.000,C 180.000} C_DIS
LIN {X 149.991,Y 2.500,Z 51.000,A 180.000,B 0.000,C 180.000} C_DIS
LIN {X 5.009,Y 2.500,Z 51.000,A 180.000,B 0.000,C 180.000} C_DIS
LIN {X 4.830,Y 2.506,Z 51.000,A 180.000,B 0.000,C 180.000} C_DIS
LIN {X 4.827,Y 2.506,Z 51.000,A 180.000,B 0.000,C 180.000} C_DIS
LIN {X 4.651,Y 2.524,Z 51.000,A 180.000,B 0.000,C 180.000} C_DIS
LIN {X 4.472,Y 2.556,Z 51.000,A 180.000,B 0.000,C 180.000} C_DIS
LIN {X 4.294,Y 2.602,Z 51.000,A 180.000,B 0.000,C 180.000} C_DIS
LIN {X 4.115,Y 2.662,Z 51.000,A 180.000,B 0.000,C 180.000} C_DIS
LIN {X 4.057,Y 2.685,Z 51.000,A 180.000,B 0.000,C 180.000} C_DIS
LIN {X 3.936,Y 2.738,Z 51.000,A 180.000,B 0.000,C 180.000} C_DIS
LIN {X 3.757,Y 2.831,Z 51.000,A 180.000,B 0.000,C 180.000} C_DIS
LIN {X 3.702,Y 2.864,Z 51.000,A 180.000,B 0.000,C 180.000} C_DIS
LIN {X 3.579,Y 2.943,Z 51.000,A 180.000,B 0.000,C 180.000} C_DIS
LIN {X 3.445,Y 3.042,Z 51.000,A 180.000,B 0.000,C 180.000} C_DIS
LIN {X 3.400,Y 3.079,Z 51.000,A 180.000,B 0.000,C 180.000} C_DIS
LIN {X 3.243,Y 3.221,Z 51.000,A 180.000,B 0.000,C 180.000} C_DIS
LIN {X 3.221,Y 3.243,Z 51.000,A 180.000,B 0.000,C 180.000} C_DIS
LIN {X 3.079,Y 3.400,Z 51.000,A 180.000,B 0.000,C 180.000} C_DIS
LIN {X 3.042,Y 3.445,Z 51.000,A 180.000,B 0.000,C 180.000} C_DIS
LIN {X 2.943,Y 3.579,Z 51.000,A 180.000,B 0.000,C 180.000} C_DIS
LIN {X 2.864,Y 3.702,Z 51.000,A 180.000,B 0.000,C 180.000} C_DIS
LIN {X 2.831,Y 3.757,Z 51.000,A 180.000,B 0.000,C 180.000} C_DIS
LIN {X 2.738,Y 3.936,Z 51.000,A 180.000,B 0.000,C 180.000} C_DIS
LIN {X 2.685,Y 4.057,Z 51.000,A 180.000,B 0.000,C 180.000} C_DIS
LIN {X 2.662,Y 4.115,Z 51.000,A 180.000,B 0.000,C 180.000} C_DIS
LIN {X 2.602,Y 4.294,Z 51.000,A 180.000,B 0.000,C 180.000} C_DIS
LIN {X 2.556,Y 4.472,Z 51.000,A 180.000,B 0.000,C 180.000} C_DIS
LIN {X 2.524,Y 4.651,Z 51.000,A 180.000,B 0.000,C 180.000} C_DIS
LIN {X 2.506,Y 4.827,Z 51.000,A 180.000,B 0.000,C 180.000} C_DIS
LIN {X 2.506,Y 4.830,Z 51.000,A 180.000,B 0.000,C 180.000} C_DIS
LIN {X 2.500,Y 5.009,Z 51.000,A 180.000,B 0.000,C 180.000} C_DIS
LIN {X 2.500,Y 149.991,Z 51.000,A 180.000,B 0.000,C 180.000} C_DIS
LIN {X 2.506,Y 150.170,Z 51.000,A 180.000,B 0.000,C 180.000} C_DIS
LIN {X 2.506,Y 150.173,Z 51.000,A 180.000,B 0.000,C 180.000} C_DIS
LIN {X 2.524,Y 150.349,Z 51.000,A 180.000,B 0.000,C 180.000} C_DIS
LIN {X 2.556,Y 150.528,Z 51.000,A 180.000,B 0.000,C 180.000} C_DIS
LIN {X 2.602,Y 150.706,Z 51.000,A 180.000,B 0.000,C 180.000} C_DIS
LIN {X 2.662,Y 150.885,Z 51.000,A 180.000,B 0.000,C 180.000} C_DIS
LIN {X 2.685,Y 150.943,Z 51.000,A 180.000,B 0.000,C 180.000} C_DIS
LIN {X 2.738,Y 151.064,Z 51.000,A 180.000,B 0.000,C 180.000} C_DIS
LIN {X 2.831,Y 151.243,Z 51.000,A 180.000,B 0.000,C 180.000} C_DIS
LIN {X 2.864,Y 151.298,Z 51.000,A 180.000,B 0.000,C 180.000} C_DIS
LIN {X 2.943,Y 151.421,Z 51.000,A 180.000,B 0.000,C 180.000} C_DIS
LIN {X 3.042,Y 151.555,Z 51.000,A 180.000,B 0.000,C 180.000} C_DIS
LIN {X 3.079,Y 151.600,Z 51.000,A 180.000,B 0.000,C 180.000} C_DIS
LIN {X 3.221,Y 151.757,Z 51.000,A 180.000,B 0.000,C 180.000} C_DIS
LIN {X 3.243,Y 151.779,Z 51.000,A 180.000,B 0.000,C 180.000} C_DIS
LIN {X 3.400,Y 151.921,Z 51.000,A 180.000,B 0.000,C 180.000} C_DIS
LIN {X 3.445,Y 151.958,Z 51.000,A 180.000,B 0.000,C 180.000} C_DIS
LIN {X 3.579,Y 152.057,Z 51.000,A 180.000,B 0.000,C 180.000} C_DIS
LIN {X 3.702,Y 152.136,Z 51.000,A 180.000,B 0.000,C 180.000} C_DIS
LIN {X 3.757,Y 152.169,Z 51.000,A 180.000,B 0.000,C 180.000} C_DIS
LIN {X 3.936,Y 152.262,Z 51.000,A 180.000,B 0.000,C 180.000} C_DIS
LIN {X 4.057,Y 152.315,Z 51.000,A 180.000,B 0.000,C 180.000} C_DIS
LIN {X 4.115,Y 152.338,Z 51.000,A 180.000,B 0.000,C 180.000} C_DIS
LIN {X 4.294,Y 152.398,Z 51.000,A 180.000,B 0.000,C 180.000} C_DIS
LIN {X 4.472,Y 152.444,Z 51.000,A 180.000,B 0.000,C 180.000} C_DIS
LIN {X 4.651,Y 152.476,Z 51.000,A 180.000,B 0.000,C 180.000} C_DIS
LIN {X 4.827,Y 152.494,Z 51.000,A 180.000,B 0.000,C 180.000} C_DIS
LIN {X 4.830,Y 152.494,Z 51.000,A 180.000,B 0.000,C 180.000} C_DIS
LIN {X 5.009,Y 152.500,Z 51.000,A 180.000,B 0.000,C 180.000} C_DIS
LIN {X 149.991,Y 152.500,Z 51.000,A 180.000,B 0.000,C 180.000} C_DIS
LIN {X 150.170,Y 152.494,Z 51.000,A 180.000,B 0.000,C 180.000} C_DIS
LIN {X 150.173,Y 152.494,Z 51.000,A 180.000,B 0.000,C 180.000} C_DIS
LIN {X 150.349,Y 152.476,Z 51.000,A 180.000,B 0.000,C 180.000} C_DIS
LIN {X 150.528,Y 152.444,Z 51.000,A 180.000,B 0.000,C 180.000} C_DIS
LIN {X 150.706,Y 152.398,Z 51.000,A 180.000,B 0.000,C 180.000} C_DIS
LIN {X 150.885,Y 152.338,Z 51.000,A 180.000,B 0.000,C 180.000} C_DIS
LIN {X 150.943,Y 152.315,Z 51.000,A 180.000,B 0.000,C 180.000} C_DIS
LIN {X 151.064,Y 152.262,Z 51.000,A 180.000,B 0.000,C 180.000} C_DIS
LIN {X 151.243,Y 152.169,Z 51.000,A 180.000,B 0.000,C 180.000} C_DIS
LIN {X 151.298,Y 152.136,Z 51.000,A 180.000,B 0.000,C 180.000} C_DIS
LIN {X 151.421,Y 152.057,Z 51.000,A 180.000,B 0.000,C 180.000} C_DIS
LIN {X 151.555,Y 151.958,Z 51.000,A 180.000,B 0.000,C 180.000} C_DIS
LIN {X 151.600,Y 151.921,Z 51.000,A 180.000,B 0.000,C 180.000} C_DIS
LIN {X 151.757,Y 151.779,Z 51.000,A 180.000,B 0.000,C 180.000} C_DIS
LIN {X 151.779,Y 151.757,Z 51.000,A 180.000,B 0.000,C 180.000} C_DIS
LIN {X 151.921,Y 151.600,Z 51.000,A 180.000,B 0.000,C 180.000} C_DIS
LIN {X 151.958,Y 151.555,Z 51.000,A 180.000,B 0.000,C 180.000} C_DIS
LIN {X 152.057,Y 151.421,Z 51.000,A 180.000,B 0.000,C 180.000} C_DIS
LIN {X 152.136,Y 151.298,Z 51.000,A 180.000,B 0.000,C 180.000} C_DIS
LIN {X 152.169,Y 151.243,Z 51.000,A 180.000,B 0.000,C 180.000} C_DIS
LIN {X 152.262,Y 151.064,Z 51.000,A 180.000,B 0.000,C 180.000} C_DIS
LIN {X 152.315,Y 150.943,Z 51.000,A 180.000,B 0.000,C 180.000} C_DIS
LIN {X 152.338,Y 150.885,Z 51.000,A 180.000,B 0.000,C 180.000} C_DIS
LIN {X 152.398,Y 150.706,Z 51.000,A 180.000,B 0.000,C 180.000} C_DIS
LIN {X 152.444,Y 150.528,Z 51.000,A 180.000,B 0.000,C 180.000} C_DIS
LIN {X 152.476,Y 150.349,Z 51.000,A 180.000,B 0.000,C 180.000} C_DIS
LIN {X 152.494,Y 150.173,Z 51.000,A 180.000,B 0.000,C 180.000} C_DIS
LIN {X 152.494,Y 150.170,Z 51.000,A 180.000,B 0.000,C 180.000} C_DIS
LIN {X 152.500,Y 149.991,Z 51.000,A 180.000,B 0.000,C 180.000} C_DIS
LIN {X 152.500,Y 72.697,Z 51.000,A 180.000,B 0.000,C 180.000} C_DIS
; Link Move Starts
LIN {X 152.500,Y 72.382,Z 51.000,A 180.000,B 0.000,C 180.000} C_DIS
LIN {X 152.500,Y 72.067,Z 50.999,A 180.000,B 0.000,C 180.000} C_DIS
LIN {X 152.500,Y 71.752,Z 50.998,A 180.000,B 0.000,C 180.000} C_DIS
LIN {X 152.500,Y 71.437,Z 50.996,A 180.000,B 0.000,C 180.000} C_DIS
LIN {X 152.500,Y 71.122,Z 50.994,A 180.000,B 0.000,C 180.000} C_DIS
LIN {X 152.500,Y 70.807,Z 50.991,A 180.000,B 0.000,C 180.000} C_DIS
LIN {X 152.500,Y 70.492,Z 50.988,A 180.000,B 0.000,C 180.000} C_DIS
LIN {X 152.500,Y 70.177,Z 50.985,A 180.000,B 0.000,C 180.000} C_DIS
LIN {X 152.500,Y 69.862,Z 50.981,A 180.000,B 0.000,C 180.000} C_DIS
LIN {X 152.500,Y 69.547,Z 50.977,A 180.000,B 0.000,C 180.000} C_DIS
LIN {X 152.500,Y 69.232,Z 50.972,A 180.000,B 0.000,C 180.000} C_DIS
LIN {X 152.500,Y 69.075,Z 50.969,A 180.000,B 0.000,C 180.000} C_DIS
LIN {X 152.500,Y 68.917,Z 50.967,A 180.000,B 0.000,C 180.000} C_DIS
LIN {X 152.500,Y 68.760,Z 50.964,A 180.000,B 0.000,C 180.000} C_DIS
LIN {X 152.500,Y 68.602,Z 50.961,A 180.000,B 0.000,C 180.000} C_DIS
LIN {X 152.500,Y 68.445,Z 50.959,A 180.000,B 0.000,C 180.000} C_DIS
LIN {X 152.500,Y 68.287,Z 50.956,A 180.000,B 0.000,C 180.000} C_DIS
LIN {X 152.500,Y 68.130,Z 50.952,A 180.000,B 0.000,C 180.000} C_DIS
LIN {X 152.500,Y 67.972,Z 50.949,A 180.000,B 0.000,C 180.000} C_DIS
LIN {X 152.500,Y 67.815,Z 50.946,A 180.000,B 0.000,C 180.000} C_DIS
LIN {X 152.500,Y 67.657,Z 50.943,A 180.000,B 0.000,C 180.000} C_DIS
LIN {X 152.500,Y 67.500,Z 50.939,A 180.000,B 0.000,C 180.000} C_DIS
LIN {X 152.500,Y 67.342,Z 50.936,A 180.000,B 0.000,C 180.000} C_DIS
LIN {X 152.500,Y 67.185,Z 50.932,A 180.000,B 0.000,C 180.000} C_DIS
LIN {X 152.500,Y 67.027,Z 50.928,A 180.000,B 0.000,C 180.000} C_DIS
LIN {X 152.500,Y 66.870,Z 50.925,A 180.000,B 0.000,C 180.000} C_DIS
LIN {X 152.500,Y 66.712,Z 50.921,A 180.000,B 0.000,C 180.000} C_DIS
LIN {X 152.500,Y 66.555,Z 50.917,A 180.000,B 0.000,C 180.000} C_DIS
LIN {X 152.500,Y 66.397,Z 50.913,A 180.000,B 0.000,C 180.000} C_DIS
LIN {X 152.500,Y 66.240,Z 50.909,A 180.000,B 0.000,C 180.000} C_DIS
LIN {X 152.500,Y 66.082,Z 50.905,A 180.000,B 0.000,C 180.000} C_DIS
LIN {X 152.500,Y 65.925,Z 50.900,A 180.000,B 0.000,C 180.000} C_DIS
LIN {X 152.500,Y 65.767,Z 50.896,A 180.000,B 0.000,C 180.000} C_DIS
LIN {X 152.500,Y 65.610,Z 50.892,A 180.000,B 0.000,C 180.000} C_DIS
LIN {X 152.500,Y 65.452,Z 50.887,A 180.000,B 0.000,C 180.000} C_DIS
LIN {X 152.500,Y 65.295,Z 50.883,A 180.000,B 0.000,C 180.000} C_DIS
LIN {X 152.500,Y 65.137,Z 50.878,A 180.000,B 0.000,C 180.000} C_DIS
LIN {X 152.500,Y 64.980,Z 50.873,A 180.000,B 0.000,C 180.000} C_DIS
LIN {X 152.500,Y 64.822,Z 50.869,A 180.000,B 0.000,C 180.000} C_DIS
LIN {X 152.500,Y 64.665,Z 50.864,A 180.000,B 0.000,C 180.000} C_DIS
LIN {X 152.500,Y 64.507,Z 50.859,A 180.000,B 0.000,C 180.000} C_DIS
LIN {X 152.500,Y 64.350,Z 50.854,A 180.000,B 0.000,C 180.000} C_DIS
LIN {X 152.500,Y 64.271,Z 50.851,A 180.000,B 0.000,C 180.000} C_DIS
LIN {X 152.500,Y 64.192,Z 50.849,A 180.000,B 0.000,C 180.000} C_DIS
LIN {X 152.500,Y 64.113,Z 50.846,A 180.000,B 0.000,C 180.000} C_DIS
LIN {X 152.500,Y 64.035,Z 50.844,A 180.000,B 0.000,C 180.000} C_DIS
LIN {X 152.500,Y 63.956,Z 50.841,A 180.000,B 0.000,C 180.000} C_DIS
LIN {X 152.500,Y 63.877,Z 50.839,A 180.000,B 0.000,C 180.000} C_DIS
LIN {X 152.500,Y 63.798,Z 50.836,A 180.000,B 0.000,C 180.000} C_DIS
LIN {X 152.500,Y 63.641,Z 50.831,A 180.000,B 0.000,C 180.000} C_DIS
LIN {X 152.500,Y 63.483,Z 50.825,A 180.000,B 0.000,C 180.000} C_DIS
LIN {X 152.500,Y 63.326,Z 50.820,A 180.000,B 0.000,C 180.000} C_DIS
LIN {X 152.500,Y 63.168,Z 50.815,A 180.000,B 0.000,C 180.000} C_DIS
LIN {X 152.500,Y 63.011,Z 50.809,A 180.000,B 0.000,C 180.000} C_DIS
LIN {X 152.500,Y 62.932,Z 50.806,A 180.000,B 0.000,C 180.000} C_DIS
LIN {X 152.500,Y 62.775,Z 50.801,A 180.000,B 0.000,C 180.000} C_DIS
LIN {X 152.500,Y 62.538,Z 50.793,A 180.000,B 0.000,C 180.000} C_DIS
LIN {X 152.500,Y 62.381,Z 50.787,A 180.000,B 0.000,C 180.000} C_DIS
LIN {X 152.500,Y 62.302,Z 50.785,A 180.000,B 0.000,C 180.000} C_DIS
LIN {X 152.500,Y 62.145,Z 50.779,A 180.000,B 0.000,C 180.000} C_DIS
LIN {X 152.500,Y 61.908,Z 50.771,A 180.000,B 0.000,C 180.000} C_DIS
LIN {X 152.500,Y 61.751,Z 50.765,A 180.000,B 0.000,C 180.000} C_DIS
LIN {X 152.500,Y 61.672,Z 50.763,A 180.000,B 0.000,C 180.000} C_DIS
LIN {X 152.500,Y 61.515,Z 50.757,A 180.000,B 0.000,C 180.000} C_DIS
LIN {X 152.500,Y 61.278,Z 50.749,A 180.000,B 0.000,C 180.000} C_DIS
LIN {X 152.500,Y 61.121,Z 50.743,A 180.000,B 0.000,C 180.000} C_DIS
LIN {X 152.500,Y 61.042,Z 50.741,A 180.000,B 0.000,C 180.000} C_DIS
LIN {X 152.500,Y 60.885,Z 50.735,A 180.000,B 0.000,C 180.000} C_DIS
LIN {X 152.500,Y 60.648,Z 50.727,A 180.000,B 0.000,C 180.000} C_DIS
LIN {X 152.500,Y 60.491,Z 50.721,A 180.000,B 0.000,C 180.000} C_DIS
LIN {X 152.500,Y 60.412,Z 50.719,A 180.000,B 0.000,C 180.000} C_DIS
LIN {X 152.500,Y 60.255,Z 50.713,A 180.000,B 0.000,C 180.000} C_DIS
LIN {X 152.500,Y 59.782,Z 50.697,A 180.000,B 0.000,C 180.000} C_DIS
LIN {X 152.500,Y 59.625,Z 50.691,A 180.000,B 0.000,C 180.000} C_DIS
LIN {X 152.500,Y 59.152,Z 50.675,A 180.000,B 0.000,C 180.000} C_DIS
LIN {X 152.500,Y 58.995,Z 50.669,A 180.000,B 0.000,C 180.000} C_DIS
LIN {X 152.500,Y 58.443,Z 50.650,A 180.000,B 0.000,C 180.000} C_DIS
LIN {X 152.500,Y 57.971,Z 50.633,A 180.000,B 0.000,C 180.000} C_DIS
LIN {X 152.500,Y 57.813,Z 50.628,A 180.000,B 0.000,C 180.000} C_DIS
LIN {X 152.500,Y 57.341,Z 50.611,A 180.000,B 0.000,C 180.000} C_DIS
LIN {X 152.500,Y 57.183,Z 50.606,A 180.000,B 0.000,C 180.000} C_DIS
LIN {X 152.500,Y 56.396,Z 50.578,A 180.000,B 0.000,C 180.000} C_DIS
LIN {X 152.500,Y 56.002,Z 50.565,A 180.000,B 0.000,C 180.000} C_DIS
LIN {X 152.500,Y 55.530,Z 50.548,A 180.000,B 0.000,C 180.000} C_DIS
LIN {X 152.500,Y 53.718,Z 50.485,A 180.000,B 0.000,C 180.000} C_DIS
LIN {X 152.500,Y 50.726,Z 50.380,A 180.000,B 0.000,C 180.000} C_DIS
LIN {X 152.500,Y 50.568,Z 50.375,A 180.000,B 0.000,C 180.000} C_DIS
LIN {X 152.500,Y 50.096,Z 50.358,A 180.000,B 0.000,C 180.000} C_DIS
LIN {X 152.500,Y 49.938,Z 50.353,A 180.000,B 0.000,C 180.000} C_DIS
LIN {X 152.500,Y 49.466,Z 50.336,A 180.000,B 0.000,C 180.000} C_DIS
LIN {X 152.500,Y 49.387,Z 50.334,A 180.000,B 0.000,C 180.000} C_DIS
LIN {X 152.500,Y 49.230,Z 50.328,A 180.000,B 0.000,C 180.000} C_DIS
LIN {X 152.500,Y 48.757,Z 50.312,A 180.000,B 0.000,C 180.000} C_DIS
LIN {X 152.500,Y 48.600,Z 50.306,A 180.000,B 0.000,C 180.000} C_DIS
LIN {X 152.500,Y 48.127,Z 50.290,A 180.000,B 0.000,C 180.000} C_DIS
LIN {X 152.500,Y 47.970,Z 50.284,A 180.000,B 0.000,C 180.000} C_DIS
LIN {X 152.500,Y 47.733,Z 50.276,A 180.000,B 0.000,C 180.000} C_DIS
LIN {X 152.500,Y 47.576,Z 50.270,A 180.000,B 0.000,C 180.000} C_DIS
LIN {X 152.500,Y 47.497,Z 50.268,A 180.000,B 0.000,C 180.000} C_DIS
LIN {X 152.500,Y 47.340,Z 50.262,A 180.000,B 0.000,C 180.000} C_DIS
LIN {X 152.500,Y 47.104,Z 50.254,A 180.000,B 0.000,C 180.000} C_DIS
LIN {X 152.500,Y 46.946,Z 50.248,A 180.000,B 0.000,C 180.000} C_DIS
LIN {X 152.500,Y 46.867,Z 50.246,A 180.000,B 0.000,C 180.000} C_DIS
LIN {X 152.500,Y 46.710,Z 50.240,A 180.000,B 0.000,C 180.000} C_DIS
LIN {X 152.500,Y 46.474,Z 50.232,A 180.000,B 0.000,C 180.000} C_DIS
LIN {X 152.500,Y 46.316,Z 50.226,A 180.000,B 0.000,C 180.000} C_DIS
LIN {X 152.500,Y 46.237,Z 50.224,A 180.000,B 0.000,C 180.000} C_DIS
LIN {X 152.500,Y 46.080,Z 50.218,A 180.000,B 0.000,C 180.000} C_DIS
LIN {X 152.500,Y 45.844,Z 50.210,A 180.000,B 0.000,C 180.000} C_DIS
LIN {X 152.500,Y 45.686,Z 50.204,A 180.000,B 0.000,C 180.000} C_DIS
LIN {X 152.500,Y 45.607,Z 50.202,A 180.000,B 0.000,C 180.000} C_DIS
LIN {X 152.500,Y 45.450,Z 50.196,A 180.000,B 0.000,C 180.000} C_DIS
LIN {X 152.500,Y 45.292,Z 50.191,A 180.000,B 0.000,C 180.000} C_DIS
LIN {X 152.500,Y 45.135,Z 50.185,A 180.000,B 0.000,C 180.000} C_DIS
LIN {X 152.500,Y 44.977,Z 50.180,A 180.000,B 0.000,C 180.000} C_DIS
LIN {X 152.500,Y 44.820,Z 50.174,A 180.000,B 0.000,C 180.000} C_DIS
LIN {X 152.500,Y 44.662,Z 50.169,A 180.000,B 0.000,C 180.000} C_DIS
LIN {X 152.500,Y 44.505,Z 50.164,A 180.000,B 0.000,C 180.000} C_DIS
LIN {X 152.500,Y 44.426,Z 50.161,A 180.000,B 0.000,C 180.000} C_DIS
LIN {X 152.500,Y 44.347,Z 50.159,A 180.000,B 0.000,C 180.000} C_DIS
LIN {X 152.500,Y 44.269,Z 50.156,A 180.000,B 0.000,C 180.000} C_DIS
LIN {X 152.500,Y 44.190,Z 50.154,A 180.000,B 0.000,C 180.000} C_DIS
LIN {X 152.500,Y 44.111,Z 50.151,A 180.000,B 0.000,C 180.000} C_DIS
LIN {X 152.500,Y 44.032,Z 50.148,A 180.000,B 0.000,C 180.000} C_DIS
LIN {X 152.500,Y 43.875,Z 50.143,A 180.000,B 0.000,C 180.000} C_DIS
LIN {X 152.500,Y 43.717,Z 50.139,A 180.000,B 0.000,C 180.000} C_DIS
LIN {X 152.500,Y 43.560,Z 50.134,A 180.000,B 0.000,C 180.000} C_DIS
LIN {X 152.500,Y 43.402,Z 50.129,A 180.000,B 0.000,C 180.000} C_DIS
LIN {X 152.500,Y 43.245,Z 50.124,A 180.000,B 0.000,C 180.000} C_DIS
LIN {X 152.500,Y 43.087,Z 50.120,A 180.000,B 0.000,C 180.000} C_DIS
LIN {X 152.500,Y 42.930,Z 50.115,A 180.000,B 0.000,C 180.000} C_DIS
LIN {X 152.500,Y 42.772,Z 50.110,A 180.000,B 0.000,C 180.000} C_DIS
LIN {X 152.500,Y 42.615,Z 50.106,A 180.000,B 0.000,C 180.000} C_DIS
LIN {X 152.500,Y 42.457,Z 50.102,A 180.000,B 0.000,C 180.000} C_DIS
LIN {X 152.500,Y 42.300,Z 50.097,A 180.000,B 0.000,C 180.000} C_DIS
LIN {X 152.500,Y 42.142,Z 50.093,A 180.000,B 0.000,C 180.000} C_DIS
LIN {X 152.500,Y 41.985,Z 50.089,A 180.000,B 0.000,C 180.000} C_DIS
LIN {X 152.500,Y 41.827,Z 50.085,A 180.000,B 0.000,C 180.000} C_DIS
LIN {X 152.500,Y 41.670,Z 50.081,A 180.000,B 0.000,C 180.000} C_DIS
LIN {X 152.500,Y 41.512,Z 50.077,A 180.000,B 0.000,C 180.000} C_DIS
LIN {X 152.500,Y 41.355,Z 50.073,A 180.000,B 0.000,C 180.000} C_DIS
LIN {X 152.500,Y 41.197,Z 50.070,A 180.000,B 0.000,C 180.000} C_DIS
LIN {X 152.500,Y 41.040,Z 50.066,A 180.000,B 0.000,C 180.000} C_DIS
LIN {X 152.500,Y 40.882,Z 50.062,A 180.000,B 0.000,C 180.000} C_DIS
LIN {X 152.500,Y 40.725,Z 50.059,A 180.000,B 0.000,C 180.000} C_DIS
LIN {X 152.500,Y 40.567,Z 50.056,A 180.000,B 0.000,C 180.000} C_DIS
LIN {X 152.500,Y 40.410,Z 50.052,A 180.000,B 0.000,C 180.000} C_DIS
LIN {X 152.500,Y 40.252,Z 50.049,A 180.000,B 0.000,C 180.000} C_DIS
LIN {X 152.500,Y 40.095,Z 50.046,A 180.000,B 0.000,C 180.000} C_DIS
LIN {X 152.500,Y 39.937,Z 50.043,A 180.000,B 0.000,C 180.000} C_DIS
LIN {X 152.500,Y 39.780,Z 50.040,A 180.000,B 0.000,C 180.000} C_DIS
LIN {X 152.500,Y 39.622,Z 50.037,A 180.000,B 0.000,C 180.000} C_DIS
LIN {X 152.500,Y 39.465,Z 50.034,A 180.000,B 0.000,C 180.000} C_DIS
LIN {X 152.500,Y 39.307,Z 50.032,A 180.000,B 0.000,C 180.000} C_DIS
LIN {X 152.500,Y 39.150,Z 50.029,A 180.000,B 0.000,C 180.000} C_DIS
LIN {X 152.500,Y 38.992,Z 50.027,A 180.000,B 0.000,C 180.000} C_DIS
LIN {X 152.500,Y 38.677,Z 50.022,A 180.000,B 0.000,C 180.000} C_DIS
LIN {X 152.500,Y 38.362,Z 50.018,A 180.000,B 0.000,C 180.000} C_DIS
LIN {X 152.500,Y 38.047,Z 50.014,A 180.000,B 0.000,C 180.000} C_DIS
LIN {X 152.500,Y 37.732,Z 50.011,A 180.000,B 0.000,C 180.000} C_DIS
LIN {X 152.500,Y 37.417,Z 50.008,A 180.000,B 0.000,C 180.000} C_DIS
LIN {X 152.500,Y 37.102,Z 50.005,A 180.000,B 0.000,C 180.000} C_DIS
LIN {X 152.500,Y 36.787,Z 50.003,A 180.000,B 0.000,C 180.000} C_DIS
LIN {X 152.500,Y 36.472,Z 50.002,A 180.000,B 0.000,C 180.000} C_DIS
LIN {X 152.500,Y 36.157,Z 50.001,A 180.000,B 0.000,C 180.000} C_DIS
LIN {X 152.500,Y 35.842,Z 50.000,A 180.000,B 0.000,C 180.000} C_DIS
LIN {X 152.500,Y 35.611,Z 50.000,A 180.000,B 0.000,C 180.000} C_DIS
; Cutting Move Starts
LIN {X 152.500,Y 5.009,Z 50.000,A 180.000,B 0.000,C 180.000} C_DIS
LIN {X 152.494,Y 4.830,Z 50.000,A 180.000,B 0.000,C 180.000} C_DIS
LIN {X 152.494,Y 4.827,Z 50.000,A 180.000,B 0.000,C 180.000} C_DIS
LIN {X 152.476,Y 4.651,Z 50.000,A 180.000,B 0.000,C 180.000} C_DIS
LIN {X 152.444,Y 4.472,Z 50.000,A 180.000,B 0.000,C 180.000} C_DIS
LIN {X 152.398,Y 4.294,Z 50.000,A 180.000,B 0.000,C 180.000} C_DIS
LIN {X 152.338,Y 4.115,Z 50.000,A 180.000,B 0.000,C 180.000} C_DIS
LIN {X 152.315,Y 4.057,Z 50.000,A 180.000,B 0.000,C 180.000} C_DIS
LIN {X 152.262,Y 3.936,Z 50.000,A 180.000,B 0.000,C 180.000} C_DIS
LIN {X 152.169,Y 3.757,Z 50.000,A 180.000,B 0.000,C 180.000} C_DIS
LIN {X 152.136,Y 3.702,Z 50.000,A 180.000,B 0.000,C 180.000} C_DIS
LIN {X 152.057,Y 3.579,Z 50.000,A 180.000,B 0.000,C 180.000} C_DIS
LIN {X 151.958,Y 3.445,Z 50.000,A 180.000,B 0.000,C 180.000} C_DIS
LIN {X 151.921,Y 3.400,Z 50.000,A 180.000,B 0.000,C 180.000} C_DIS
LIN {X 151.779,Y 3.243,Z 50.000,A 180.000,B 0.000,C 180.000} C_DIS
LIN {X 151.757,Y 3.221,Z 50.000,A 180.000,B 0.000,C 180.000} C_DIS
LIN {X 151.600,Y 3.079,Z 50.000,A 180.000,B 0.000,C 180.000} C_DIS
LIN {X 151.555,Y 3.042,Z 50.000,A 180.000,B 0.000,C 180.000} C_DIS
LIN {X 151.421,Y 2.943,Z 50.000,A 180.000,B 0.000,C 180.000} C_DIS
LIN {X 151.298,Y 2.864,Z 50.000,A 180.000,B 0.000,C 180.000} C_DIS
LIN {X 151.243,Y 2.831,Z 50.000,A 180.000,B 0.000,C 180.000} C_DIS
LIN {X 151.064,Y 2.738,Z 50.000,A 180.000,B 0.000,C 180.000} C_DIS
LIN {X 150.943,Y 2.685,Z 50.000,A 180.000,B 0.000,C 180.000} C_DIS
LIN {X 150.885,Y 2.662,Z 50.000,A 180.000,B 0.000,C 180.000} C_DIS
LIN {X 150.706,Y 2.602,Z 50.000,A 180.000,B 0.000,C 180.000} C_DIS
LIN {X 150.528,Y 2.556,Z 50.000,A 180.000,B 0.000,C 180.000} C_DIS
LIN {X 150.349,Y 2.524,Z 50.000,A 180.000,B 0.000,C 180.000} C_DIS
LIN {X 150.173,Y 2.506,Z 50.000,A 180.000,B 0.000,C 180.000} C_DIS
LIN {X 150.170,Y 2.506,Z 50.000,A 180.000,B 0.000,C 180.000} C_DIS
LIN {X 149.991,Y 2.500,Z 50.000,A 180.000,B 0.000,C 180.000} C_DIS
LIN {X 5.009,Y 2.500,Z 50.000,A 180.000,B 0.000,C 180.000} C_DIS
LIN {X 4.830,Y 2.506,Z 50.000,A 180.000,B 0.000,C 180.000} C_DIS
LIN {X 4.827,Y 2.506,Z 50.000,A 180.000,B 0.000,C 180.000} C_DIS
LIN {X 4.651,Y 2.524,Z 50.000,A 180.000,B 0.000,C 180.000} C_DIS
LIN {X 4.472,Y 2.556,Z 50.000,A 180.000,B 0.000,C 180.000} C_DIS
LIN {X 4.294,Y 2.602,Z 50.000,A 180.000,B 0.000,C 180.000} C_DIS
LIN {X 4.115,Y 2.662,Z 50.000,A 180.000,B 0.000,C 180.000} C_DIS
LIN {X 4.057,Y 2.685,Z 50.000,A 180.000,B 0.000,C 180.000} C_DIS
LIN {X 3.936,Y 2.738,Z 50.000,A 180.000,B 0.000,C 180.000} C_DIS
LIN {X 3.757,Y 2.831,Z 50.000,A 180.000,B 0.000,C 180.000} C_DIS
LIN {X 3.702,Y 2.864,Z 50.000,A 180.000,B 0.000,C 180.000} C_DIS
LIN {X 3.579,Y 2.943,Z 50.000,A 180.000,B 0.000,C 180.000} C_DIS
LIN {X 3.445,Y 3.042,Z 50.000,A 180.000,B 0.000,C 180.000} C_DIS
LIN {X 3.400,Y 3.079,Z 50.000,A 180.000,B 0.000,C 180.000} C_DIS
LIN {X 3.243,Y 3.221,Z 50.000,A 180.000,B 0.000,C 180.000} C_DIS
LIN {X 3.221,Y 3.243,Z 50.000,A 180.000,B 0.000,C 180.000} C_DIS
LIN {X 3.079,Y 3.400,Z 50.000,A 180.000,B 0.000,C 180.000} C_DIS
LIN {X 3.042,Y 3.445,Z 50.000,A 180.000,B 0.000,C 180.000} C_DIS
LIN {X 2.943,Y 3.579,Z 50.000,A 180.000,B 0.000,C 180.000} C_DIS
LIN {X 2.864,Y 3.702,Z 50.000,A 180.000,B 0.000,C 180.000} C_DIS
LIN {X 2.831,Y 3.757,Z 50.000,A 180.000,B 0.000,C 180.000} C_DIS
LIN {X 2.738,Y 3.936,Z 50.000,A 180.000,B 0.000,C 180.000} C_DIS
LIN {X 2.685,Y 4.057,Z 50.000,A 180.000,B 0.000,C 180.000} C_DIS
LIN {X 2.662,Y 4.115,Z 50.000,A 180.000,B 0.000,C 180.000} C_DIS
LIN {X 2.602,Y 4.294,Z 50.000,A 180.000,B 0.000,C 180.000} C_DIS
LIN {X 2.556,Y 4.472,Z 50.000,A 180.000,B 0.000,C 180.000} C_DIS
LIN {X 2.524,Y 4.651,Z 50.000,A 180.000,B 0.000,C 180.000} C_DIS
LIN {X 2.506,Y 4.827,Z 50.000,A 180.000,B 0.000,C 180.000} C_DIS
LIN {X 2.506,Y 4.830,Z 50.000,A 180.000,B 0.000,C 180.000} C_DIS
LIN {X 2.500,Y 5.009,Z 50.000,A 180.000,B 0.000,C 180.000} C_DIS
LIN {X 2.500,Y 149.991,Z 50.000,A 180.000,B 0.000,C 180.000} C_DIS
LIN {X 2.506,Y 150.170,Z 50.000,A 180.000,B 0.000,C 180.000} C_DIS
LIN {X 2.506,Y 150.173,Z 50.000,A 180.000,B 0.000,C 180.000} C_DIS
LIN {X 2.524,Y 150.349,Z 50.000,A 180.000,B 0.000,C 180.000} C_DIS
LIN {X 2.556,Y 150.528,Z 50.000,A 180.000,B 0.000,C 180.000} C_DIS
LIN {X 2.602,Y 150.706,Z 50.000,A 180.000,B 0.000,C 180.000} C_DIS
LIN {X 2.662,Y 150.885,Z 50.000,A 180.000,B 0.000,C 180.000} C_DIS
LIN {X 2.685,Y 150.943,Z 50.000,A 180.000,B 0.000,C 180.000} C_DIS
LIN {X 2.738,Y 151.064,Z 50.000,A 180.000,B 0.000,C 180.000} C_DIS
LIN {X 2.831,Y 151.243,Z 50.000,A 180.000,B 0.000,C 180.000} C_DIS
LIN {X 2.864,Y 151.298,Z 50.000,A 180.000,B 0.000,C 180.000} C_DIS
LIN {X 2.943,Y 151.421,Z 50.000,A 180.000,B 0.000,C 180.000} C_DIS
LIN {X 3.042,Y 151.555,Z 50.000,A 180.000,B 0.000,C 180.000} C_DIS
LIN {X 3.079,Y 151.600,Z 50.000,A 180.000,B 0.000,C 180.000} C_DIS
LIN {X 3.221,Y 151.757,Z 50.000,A 180.000,B 0.000,C 180.000} C_DIS
LIN {X 3.243,Y 151.779,Z 50.000,A 180.000,B 0.000,C 180.000} C_DIS
LIN {X 3.400,Y 151.921,Z 50.000,A 180.000,B 0.000,C 180.000} C_DIS
LIN {X 3.445,Y 151.958,Z 50.000,A 180.000,B 0.000,C 180.000} C_DIS
LIN {X 3.579,Y 152.057,Z 50.000,A 180.000,B 0.000,C 180.000} C_DIS
LIN {X 3.702,Y 152.136,Z 50.000,A 180.000,B 0.000,C 180.000} C_DIS
LIN {X 3.757,Y 152.169,Z 50.000,A 180.000,B 0.000,C 180.000} C_DIS
LIN {X 3.936,Y 152.262,Z 50.000,A 180.000,B 0.000,C 180.000} C_DIS
LIN {X 4.057,Y 152.315,Z 50.000,A 180.000,B 0.000,C 180.000} C_DIS
LIN {X 4.115,Y 152.338,Z 50.000,A 180.000,B 0.000,C 180.000} C_DIS
LIN {X 4.294,Y 152.398,Z 50.000,A 180.000,B 0.000,C 180.000} C_DIS
LIN {X 4.472,Y 152.444,Z 50.000,A 180.000,B 0.000,C 180.000} C_DIS
LIN {X 4.651,Y 152.476,Z 50.000,A 180.000,B 0.000,C 180.000} C_DIS
LIN {X 4.827,Y 152.494,Z 50.000,A 180.000,B 0.000,C 180.000} C_DIS
LIN {X 4.830,Y 152.494,Z 50.000,A 180.000,B 0.000,C 180.000} C_DIS
LIN {X 5.009,Y 152.500,Z 50.000,A 180.000,B 0.000,C 180.000} C_DIS
LIN {X 149.991,Y 152.500,Z 50.000,A 180.000,B 0.000,C 180.000} C_DIS
LIN {X 150.170,Y 152.494,Z 50.000,A 180.000,B 0.000,C 180.000} C_DIS
LIN {X 150.173,Y 152.494,Z 50.000,A 180.000,B 0.000,C 180.000} C_DIS
LIN {X 150.349,Y 152.476,Z 50.000,A 180.000,B 0.000,C 180.000} C_DIS
LIN {X 150.528,Y 152.444,Z 50.000,A 180.000,B 0.000,C 180.000} C_DIS
LIN {X 150.706,Y 152.398,Z 50.000,A 180.000,B 0.000,C 180.000} C_DIS
LIN {X 150.885,Y 152.338,Z 50.000,A 180.000,B 0.000,C 180.000} C_DIS
LIN {X 150.943,Y 152.315,Z 50.000,A 180.000,B 0.000,C 180.000} C_DIS
LIN {X 151.064,Y 152.262,Z 50.000,A 180.000,B 0.000,C 180.000} C_DIS
LIN {X 151.243,Y 152.169,Z 50.000,A 180.000,B 0.000,C 180.000} C_DIS
LIN {X 151.298,Y 152.136,Z 50.000,A 180.000,B 0.000,C 180.000} C_DIS
LIN {X 151.421,Y 152.057,Z 50.000,A 180.000,B 0.000,C 180.000} C_DIS
LIN {X 151.555,Y 151.958,Z 50.000,A 180.000,B 0.000,C 180.000} C_DIS
LIN {X 151.600,Y 151.921,Z 50.000,A 180.000,B 0.000,C 180.000} C_DIS
LIN {X 151.757,Y 151.779,Z 50.000,A 180.000,B 0.000,C 180.000} C_DIS
LIN {X 151.779,Y 151.757,Z 50.000,A 180.000,B 0.000,C 180.000} C_DIS
LIN {X 151.921,Y 151.600,Z 50.000,A 180.000,B 0.000,C 180.000} C_DIS
LIN {X 151.958,Y 151.555,Z 50.000,A 180.000,B 0.000,C 180.000} C_DIS
LIN {X 152.057,Y 151.421,Z 50.000,A 180.000,B 0.000,C 180.000} C_DIS
LIN {X 152.136,Y 151.298,Z 50.000,A 180.000,B 0.000,C 180.000} C_DIS
LIN {X 152.169,Y 151.243,Z 50.000,A 180.000,B 0.000,C 180.000} C_DIS
LIN {X 152.262,Y 151.064,Z 50.000,A 180.000,B 0.000,C 180.000} C_DIS
LIN {X 152.315,Y 150.943,Z 50.000,A 180.000,B 0.000,C 180.000} C_DIS
LIN {X 152.338,Y 150.885,Z 50.000,A 180.000,B 0.000,C 180.000} C_DIS
LIN {X 152.398,Y 150.706,Z 50.000,A 180.000,B 0.000,C 180.000} C_DIS
LIN {X 152.444,Y 150.528,Z 50.000,A 180.000,B 0.000,C 180.000} C_DIS
LIN {X 152.476,Y 150.349,Z 50.000,A 180.000,B 0.000,C 180.000} C_DIS
LIN {X 152.494,Y 150.173,Z 50.000,A 180.000,B 0.000,C 180.000} C_DIS
LIN {X 152.494,Y 150.170,Z 50.000,A 180.000,B 0.000,C 180.000} C_DIS
LIN {X 152.500,Y 149.991,Z 50.000,A 180.000,B 0.000,C 180.000} C_DIS
LIN {X 152.500,Y 72.697,Z 50.000,A 180.000,B 0.000,C 180.000} C_DIS
LIN {X 152.500,Y 35.611,Z 50.000,A 180.000,B 0.000,C 180.000} C_DIS
; Link Move Starts
LIN {X 152.500,Y 35.296,Z 50.000,A 180.000,B 0.000,C 180.000} C_DIS
LIN {X 152.500,Y 34.981,Z 49.999,A 180.000,B 0.000,C 180.000} C_DIS
LIN {X 152.500,Y 34.666,Z 49.998,A 180.000,B 0.000,C 180.000} C_DIS
LIN {X 152.500,Y 34.351,Z 49.996,A 180.000,B 0.000,C 180.000} C_DIS
LIN {X 152.500,Y 34.036,Z 49.994,A 180.000,B 0.000,C 180.000} C_DIS
LIN {X 152.500,Y 33.721,Z 49.991,A 180.000,B 0.000,C 180.000} C_DIS
LIN {X 152.500,Y 33.406,Z 49.988,A 180.000,B 0.000,C 180.000} C_DIS
LIN {X 152.500,Y 33.091,Z 49.985,A 180.000,B 0.000,C 180.000} C_DIS
LIN {X 152.500,Y 32.776,Z 49.981,A 180.000,B 0.000,C 180.000} C_DIS
LIN {X 152.500,Y 32.461,Z 49.977,A 180.000,B 0.000,C 180.000} C_DIS
LIN {X 152.500,Y 32.146,Z 49.972,A 180.000,B 0.000,C 180.000} C_DIS
LIN {X 152.500,Y 31.989,Z 49.969,A 180.000,B 0.000,C 180.000} C_DIS
LIN {X 152.500,Y 31.831,Z 49.967,A 180.000,B 0.000,C 180.000} C_DIS
LIN {X 152.500,Y 31.674,Z 49.964,A 180.000,B 0.000,C 180.000} C_DIS
LIN {X 152.500,Y 31.516,Z 49.961,A 180.000,B 0.000,C 180.000} C_DIS
LIN {X 152.500,Y 31.359,Z 49.959,A 180.000,B 0.000,C 180.000} C_DIS
LIN {X 152.500,Y 31.201,Z 49.956,A 180.000,B 0.000,C 180.000} C_DIS
LIN {X 152.500,Y 31.044,Z 49.952,A 180.000,B 0.000,C 180.000} C_DIS
LIN {X 152.500,Y 30.886,Z 49.949,A 180.000,B 0.000,C 180.000} C_DIS
LIN {X 152.500,Y 30.729,Z 49.946,A 180.000,B 0.000,C 180.000} C_DIS
LIN {X 152.500,Y 30.571,Z 49.943,A 180.000,B 0.000,C 180.000} C_DIS
LIN {X 152.500,Y 30.414,Z 49.939,A 180.000,B 0.000,C 180.000} C_DIS
LIN {X 152.500,Y 30.256,Z 49.936,A 180.000,B 0.000,C 180.000} C_DIS
LIN {X 152.500,Y 30.099,Z 49.932,A 180.000,B 0.000,C 180.000} C_DIS
LIN {X 152.500,Y 29.941,Z 49.928,A 180.000,B 0.000,C 180.000} C_DIS
LIN {X 152.500,Y 29.784,Z 49.925,A 180.000,B 0.000,C 180.000} C_DIS
LIN {X 152.500,Y 29.626,Z 49.921,A 180.000,B 0.000,C 180.000} C_DIS
LIN {X 152.500,Y 29.469,Z 49.917,A 180.000,B 0.000,C 180.000} C_DIS
LIN {X 152.500,Y 29.311,Z 49.913,A 180.000,B 0.000,C 180.000} C_DIS
LIN {X 152.500,Y 29.154,Z 49.909,A 180.000,B 0.000,C 180.000} C_DIS
LIN {X 152.500,Y 28.996,Z 49.905,A 180.000,B 0.000,C 180.000} C_DIS
LIN {X 152.500,Y 28.839,Z 49.900,A 180.000,B 0.000,C 180.000} C_DIS
LIN {X 152.500,Y 28.681,Z 49.896,A 180.000,B 0.000,C 180.000} C_DIS
LIN {X 152.500,Y 28.524,Z 49.892,A 180.000,B 0.000,C 180.000} C_DIS
LIN {X 152.500,Y 28.366,Z 49.887,A 180.000,B 0.000,C 180.000} C_DIS
LIN {X 152.500,Y 28.209,Z 49.883,A 180.000,B 0.000,C 180.000} C_DIS
LIN {X 152.500,Y 28.051,Z 49.878,A 180.000,B 0.000,C 180.000} C_DIS
LIN {X 152.500,Y 27.894,Z 49.873,A 180.000,B 0.000,C 180.000} C_DIS
LIN {X 152.500,Y 27.736,Z 49.869,A 180.000,B 0.000,C 180.000} C_DIS
LIN {X 152.500,Y 27.579,Z 49.864,A 180.000,B 0.000,C 180.000} C_DIS
LIN {X 152.500,Y 27.421,Z 49.859,A 180.000,B 0.000,C 180.000} C_DIS
LIN {X 152.500,Y 27.264,Z 49.854,A 180.000,B 0.000,C 180.000} C_DIS
LIN {X 152.500,Y 27.185,Z 49.851,A 180.000,B 0.000,C 180.000} C_DIS
LIN {X 152.500,Y 27.106,Z 49.849,A 180.000,B 0.000,C 180.000} C_DIS
LIN {X 152.500,Y 27.028,Z 49.846,A 180.000,B 0.000,C 180.000} C_DIS
LIN {X 152.500,Y 26.949,Z 49.844,A 180.000,B 0.000,C 180.000} C_DIS
LIN {X 152.500,Y 26.870,Z 49.841,A 180.000,B 0.000,C 180.000} C_DIS
LIN {X 152.500,Y 26.791,Z 49.839,A 180.000,B 0.000,C 180.000} C_DIS
LIN {X 152.500,Y 26.713,Z 49.836,A 180.000,B 0.000,C 180.000} C_DIS
LIN {X 152.500,Y 26.555,Z 49.831,A 180.000,B 0.000,C 180.000} C_DIS
LIN {X 152.500,Y 26.398,Z 49.825,A 180.000,B 0.000,C 180.000} C_DIS
LIN {X 152.500,Y 26.240,Z 49.820,A 180.000,B 0.000,C 180.000} C_DIS
LIN {X 152.500,Y 26.083,Z 49.815,A 180.000,B 0.000,C 180.000} C_DIS
LIN {X 152.500,Y 25.925,Z 49.809,A 180.000,B 0.000,C 180.000} C_DIS
LIN {X 152.500,Y 25.846,Z 49.806,A 180.000,B 0.000,C 180.000} C_DIS
LIN {X 152.500,Y 25.689,Z 49.801,A 180.000,B 0.000,C 180.000} C_DIS
LIN {X 152.500,Y 25.453,Z 49.793,A 180.000,B 0.000,C 180.000} C_DIS
LIN {X 152.500,Y 25.295,Z 49.787,A 180.000,B 0.000,C 180.000} C_DIS
LIN {X 152.500,Y 25.216,Z 49.785,A 180.000,B 0.000,C 180.000} C_DIS
LIN {X 152.500,Y 25.059,Z 49.779,A 180.000,B 0.000,C 180.000} C_DIS
LIN {X 152.500,Y 24.823,Z 49.771,A 180.000,B 0.000,C 180.000} C_DIS
LIN {X 152.500,Y 24.665,Z 49.765,A 180.000,B 0.000,C 180.000} C_DIS
LIN {X 152.500,Y 24.586,Z 49.763,A 180.000,B 0.000,C 180.000} C_DIS
LIN {X 152.500,Y 24.429,Z 49.757,A 180.000,B 0.000,C 180.000} C_DIS
LIN {X 152.500,Y 24.193,Z 49.749,A 180.000,B 0.000,C 180.000} C_DIS
LIN {X 152.500,Y 24.035,Z 49.743,A 180.000,B 0.000,C 180.000} C_DIS
LIN {X 152.500,Y 23.956,Z 49.741,A 180.000,B 0.000,C 180.000} C_DIS
LIN {X 152.500,Y 23.799,Z 49.735,A 180.000,B 0.000,C 180.000} C_DIS
LIN {X 152.500,Y 23.563,Z 49.727,A 180.000,B 0.000,C 180.000} C_DIS
LIN {X 152.500,Y 23.405,Z 49.721,A 180.000,B 0.000,C 180.000} C_DIS
LIN {X 152.500,Y 23.326,Z 49.719,A 180.000,B 0.000,C 180.000} C_DIS
LIN {X 152.500,Y 23.169,Z 49.713,A 180.000,B 0.000,C 180.000} C_DIS
LIN {X 152.500,Y 22.696,Z 49.697,A 180.000,B 0.000,C 180.000} C_DIS
LIN {X 152.500,Y 22.539,Z 49.691,A 180.000,B 0.000,C 180.000} C_DIS
LIN {X 152.500,Y 22.066,Z 49.675,A 180.000,B 0.000,C 180.000} C_DIS
LIN {X 152.500,Y 21.909,Z 49.669,A 180.000,B 0.000,C 180.000} C_DIS
LIN {X 152.500,Y 21.358,Z 49.650,A 180.000,B 0.000,C 180.000} C_DIS
LIN {X 152.500,Y 20.885,Z 49.633,A 180.000,B 0.000,C 180.000} C_DIS
LIN {X 152.500,Y 20.728,Z 49.628,A 180.000,B 0.000,C 180.000} C_DIS
LIN {X 152.500,Y 20.255,Z 49.611,A 180.000,B 0.000,C 180.000} C_DIS
LIN {X 152.500,Y 20.098,Z 49.606,A 180.000,B 0.000,C 180.000} C_DIS
LIN {X 152.500,Y 19.310,Z 49.578,A 180.000,B 0.000,C 180.000} C_DIS
LIN {X 152.500,Y 18.916,Z 49.565,A 180.000,B 0.000,C 180.000} C_DIS
LIN {X 152.500,Y 18.444,Z 49.548,A 180.000,B 0.000,C 180.000} C_DIS
LIN {X 152.500,Y 16.633,Z 49.485,A 180.000,B 0.000,C 180.000} C_DIS
LIN {X 152.500,Y 13.640,Z 49.380,A 180.000,B 0.000,C 180.000} C_DIS
LIN {X 152.500,Y 13.483,Z 49.375,A 180.000,B 0.000,C 180.000} C_DIS
LIN {X 152.500,Y 13.010,Z 49.358,A 180.000,B 0.000,C 180.000} C_DIS
LIN {X 152.500,Y 12.853,Z 49.353,A 180.000,B 0.000,C 180.000} C_DIS
LIN {X 152.500,Y 12.380,Z 49.336,A 180.000,B 0.000,C 180.000} C_DIS
LIN {X 152.500,Y 12.302,Z 49.334,A 180.000,B 0.000,C 180.000} C_DIS
LIN {X 152.500,Y 12.144,Z 49.328,A 180.000,B 0.000,C 180.000} C_DIS
LIN {X 152.500,Y 11.672,Z 49.312,A 180.000,B 0.000,C 180.000} C_DIS
LIN {X 152.500,Y 11.514,Z 49.306,A 180.000,B 0.000,C 180.000} C_DIS
LIN {X 152.500,Y 11.042,Z 49.290,A 180.000,B 0.000,C 180.000} C_DIS
LIN {X 152.500,Y 10.884,Z 49.284,A 180.000,B 0.000,C 180.000} C_DIS
LIN {X 152.500,Y 10.648,Z 49.276,A 180.000,B 0.000,C 180.000} C_DIS
LIN {X 152.500,Y 10.490,Z 49.270,A 180.000,B 0.000,C 180.000} C_DIS
LIN {X 152.500,Y 10.412,Z 49.268,A 180.000,B 0.000,C 180.000} C_DIS
LIN {X 152.500,Y 10.254,Z 49.262,A 180.000,B 0.000,C 180.000} C_DIS
LIN {X 152.500,Y 10.018,Z 49.254,A 180.000,B 0.000,C 180.000} C_DIS
LIN {X 152.500,Y 9.860,Z 49.248,A 180.000,B 0.000,C 180.000} C_DIS
LIN {X 152.500,Y 9.782,Z 49.246,A 180.000,B 0.000,C 180.000} C_DIS
LIN {X 152.500,Y 9.624,Z 49.240,A 180.000,B 0.000,C 180.000} C_DIS
LIN {X 152.500,Y 9.388,Z 49.232,A 180.000,B 0.000,C 180.000} C_DIS
LIN {X 152.500,Y 9.230,Z 49.226,A 180.000,B 0.000,C 180.000} C_DIS
LIN {X 152.500,Y 9.152,Z 49.224,A 180.000,B 0.000,C 180.000} C_DIS
LIN {X 152.500,Y 8.994,Z 49.218,A 180.000,B 0.000,C 180.000} C_DIS
LIN {X 152.500,Y 8.758,Z 49.210,A 180.000,B 0.000,C 180.000} C_DIS
LIN {X 152.500,Y 8.600,Z 49.204,A 180.000,B 0.000,C 180.000} C_DIS
LIN {X 152.500,Y 8.522,Z 49.202,A 180.000,B 0.000,C 180.000} C_DIS
LIN {X 152.500,Y 8.364,Z 49.196,A 180.000,B 0.000,C 180.000} C_DIS
LIN {X 152.500,Y 8.207,Z 49.191,A 180.000,B 0.000,C 180.000} C_DIS
LIN {X 152.500,Y 8.049,Z 49.185,A 180.000,B 0.000,C 180.000} C_DIS
LIN {X 152.500,Y 7.892,Z 49.180,A 180.000,B 0.000,C 180.000} C_DIS
LIN {X 152.500,Y 7.734,Z 49.174,A 180.000,B 0.000,C 180.000} C_DIS
LIN {X 152.500,Y 7.577,Z 49.169,A 180.000,B 0.000,C 180.000} C_DIS
LIN {X 152.500,Y 7.419,Z 49.164,A 180.000,B 0.000,C 180.000} C_DIS
LIN {X 152.500,Y 7.340,Z 49.161,A 180.000,B 0.000,C 180.000} C_DIS
LIN {X 152.500,Y 7.262,Z 49.159,A 180.000,B 0.000,C 180.000} C_DIS
LIN {X 152.500,Y 7.183,Z 49.156,A 180.000,B 0.000,C 180.000} C_DIS
LIN {X 152.500,Y 7.104,Z 49.154,A 180.000,B 0.000,C 180.000} C_DIS
LIN {X 152.500,Y 7.025,Z 49.151,A 180.000,B 0.000,C 180.000} C_DIS
LIN {X 152.500,Y 6.947,Z 49.148,A 180.000,B 0.000,C 180.000} C_DIS
LIN {X 152.500,Y 6.789,Z 49.143,A 180.000,B 0.000,C 180.000} C_DIS
LIN {X 152.500,Y 6.632,Z 49.139,A 180.000,B 0.000,C 180.000} C_DIS
LIN {X 152.500,Y 6.474,Z 49.134,A 180.000,B 0.000,C 180.000} C_DIS
LIN {X 152.500,Y 6.317,Z 49.129,A 180.000,B 0.000,C 180.000} C_DIS
LIN {X 152.500,Y 6.159,Z 49.124,A 180.000,B 0.000,C 180.000} C_DIS
LIN {X 152.500,Y 6.002,Z 49.120,A 180.000,B 0.000,C 180.000} C_DIS
LIN {X 152.500,Y 5.844,Z 49.115,A 180.000,B 0.000,C 180.000} C_DIS
LIN {X 152.500,Y 5.687,Z 49.110,A 180.000,B 0.000,C 180.000} C_DIS
LIN {X 152.500,Y 5.529,Z 49.106,A 180.000,B 0.000,C 180.000} C_DIS
LIN {X 152.500,Y 5.372,Z 49.102,A 180.000,B 0.000,C 180.000} C_DIS
LIN {X 152.500,Y 5.214,Z 49.097,A 180.000,B 0.000,C 180.000} C_DIS
LIN {X 152.500,Y 5.057,Z 49.093,A 180.000,B 0.000,C 180.000} C_DIS
LIN {X 152.498,Y 4.899,Z 49.089,A 180.000,B 0.000,C 180.000} C_DIS
LIN {X 152.487,Y 4.742,Z 49.085,A 180.000,B 0.000,C 180.000} C_DIS
LIN {X 152.465,Y 4.586,Z 49.081,A 180.000,B 0.000,C 180.000} C_DIS
LIN {X 152.434,Y 4.431,Z 49.077,A 180.000,B 0.000,C 180.000} C_DIS
LIN {X 152.394,Y 4.279,Z 49.073,A 180.000,B 0.000,C 180.000} C_DIS
LIN {X 152.344,Y 4.130,Z 49.070,A 180.000,B 0.000,C 180.000} C_DIS
LIN {X 152.284,Y 3.984,Z 49.066,A 180.000,B 0.000,C 180.000} C_DIS
LIN {X 152.216,Y 3.842,Z 49.062,A 180.000,B 0.000,C 180.000} C_DIS
LIN {X 152.138,Y 3.705,Z 49.059,A 180.000,B 0.000,C 180.000} C_DIS
LIN {X 152.053,Y 3.573,Z 49.056,A 180.000,B 0.000,C 180.000} C_DIS
LIN {X 151.959,Y 3.447,Z 49.052,A 180.000,B 0.000,C 180.000} C_DIS
LIN {X 151.857,Y 3.326,Z 49.049,A 180.000,B 0.000,C 180.000} C_DIS
LIN {X 151.748,Y 3.213,Z 49.046,A 180.000,B 0.000,C 180.000} C_DIS
LIN {X 151.632,Y 3.106,Z 49.043,A 180.000,B 0.000,C 180.000} C_DIS
LIN {X 151.509,Y 3.007,Z 49.040,A 180.000,B 0.000,C 180.000} C_DIS
LIN {X 151.381,Y 2.916,Z 49.037,A 180.000,B 0.000,C 180.000} C_DIS
LIN {X 151.247,Y 2.833,Z 49.034,A 180.000,B 0.000,C 180.000} C_DIS
LIN {X 151.108,Y 2.759,Z 49.032,A 180.000,B 0.000,C 180.000} C_DIS
LIN {X 150.965,Y 2.694,Z 49.029,A 180.000,B 0.000,C 180.000} C_DIS
LIN {X 150.818,Y 2.637,Z 49.027,A 180.000,B 0.000,C 180.000} C_DIS
LIN {X 150.667,Y 2.591,Z 49.024,A 180.000,B 0.000,C 180.000} C_DIS
LIN {X 150.514,Y 2.553,Z 49.022,A 180.000,B 0.000,C 180.000} C_DIS
LIN {X 150.359,Y 2.526,Z 49.020,A 180.000,B 0.000,C 180.000} C_DIS
LIN {X 150.203,Y 2.508,Z 49.018,A 180.000,B 0.000,C 180.000} C_DIS
LIN {X 149.888,Y 2.500,Z 49.014,A 180.000,B 0.000,C 180.000} C_DIS
LIN {X 149.573,Y 2.500,Z 49.011,A 180.000,B 0.000,C 180.000} C_DIS
LIN {X 149.258,Y 2.500,Z 49.008,A 180.000,B 0.000,C 180.000} C_DIS
LIN {X 148.943,Y 2.500,Z 49.005,A 180.000,B 0.000,C 180.000} C_DIS
LIN {X 148.628,Y 2.500,Z 49.003,A 180.000,B 0.000,C 180.000} C_DIS
LIN {X 148.313,Y 2.500,Z 49.002,A 180.000,B 0.000,C 180.000} C_DIS
LIN {X 147.998,Y 2.500,Z 49.001,A 180.000,B 0.000,C 180.000} C_DIS
LIN {X 147.683,Y 2.500,Z 49.000,A 180.000,B 0.000,C 180.000} C_DIS
LIN {X 147.452,Y 2.500,Z 49.000,A 180.000,B 0.000,C 180.000} C_DIS
; Cutting Move Starts
LIN {X 5.009,Y 2.500,Z 49.000,A 180.000,B 0.000,C 180.000} C_DIS
LIN {X 4.830,Y 2.506,Z 49.000,A 180.000,B 0.000,C 180.000} C_DIS
LIN {X 4.827,Y 2.506,Z 49.000,A 180.000,B 0.000,C 180.000} C_DIS
LIN {X 4.651,Y 2.524,Z 49.000,A 180.000,B 0.000,C 180.000} C_DIS
LIN {X 4.472,Y 2.556,Z 49.000,A 180.000,B 0.000,C 180.000} C_DIS
LIN {X 4.294,Y 2.602,Z 49.000,A 180.000,B 0.000,C 180.000} C_DIS
LIN {X 4.115,Y 2.662,Z 49.000,A 180.000,B 0.000,C 180.000} C_DIS
LIN {X 4.057,Y 2.685,Z 49.000,A 180.000,B 0.000,C 180.000} C_DIS
LIN {X 3.936,Y 2.738,Z 49.000,A 180.000,B 0.000,C 180.000} C_DIS
LIN {X 3.757,Y 2.831,Z 49.000,A 180.000,B 0.000,C 180.000} C_DIS
LIN {X 3.702,Y 2.864,Z 49.000,A 180.000,B 0.000,C 180.000} C_DIS
LIN {X 3.579,Y 2.943,Z 49.000,A 180.000,B 0.000,C 180.000} C_DIS
LIN {X 3.445,Y 3.042,Z 49.000,A 180.000,B 0.000,C 180.000} C_DIS
LIN {X 3.400,Y 3.079,Z 49.000,A 180.000,B 0.000,C 180.000} C_DIS
LIN {X 3.243,Y 3.221,Z 49.000,A 180.000,B 0.000,C 180.000} C_DIS
LIN {X 3.221,Y 3.243,Z 49.000,A 180.000,B 0.000,C 180.000} C_DIS
LIN {X 3.079,Y 3.400,Z 49.000,A 180.000,B 0.000,C 180.000} C_DIS
LIN {X 3.042,Y 3.445,Z 49.000,A 180.000,B 0.000,C 180.000} C_DIS
LIN {X 2.943,Y 3.579,Z 49.000,A 180.000,B 0.000,C 180.000} C_DIS
LIN {X 2.864,Y 3.702,Z 49.000,A 180.000,B 0.000,C 180.000} C_DIS
LIN {X 2.831,Y 3.757,Z 49.000,A 180.000,B 0.000,C 180.000} C_DIS
LIN {X 2.738,Y 3.936,Z 49.000,A 180.000,B 0.000,C 180.000} C_DIS
LIN {X 2.685,Y 4.057,Z 49.000,A 180.000,B 0.000,C 180.000} C_DIS
LIN {X 2.662,Y 4.115,Z 49.000,A 180.000,B 0.000,C 180.000} C_DIS
LIN {X 2.602,Y 4.294,Z 49.000,A 180.000,B 0.000,C 180.000} C_DIS
LIN {X 2.556,Y 4.472,Z 49.000,A 180.000,B 0.000,C 180.000} C_DIS
LIN {X 2.524,Y 4.651,Z 49.000,A 180.000,B 0.000,C 180.000} C_DIS
LIN {X 2.506,Y 4.827,Z 49.000,A 180.000,B 0.000,C 180.000} C_DIS
LIN {X 2.506,Y 4.830,Z 49.000,A 180.000,B 0.000,C 180.000} C_DIS
LIN {X 2.500,Y 5.009,Z 49.000,A 180.000,B 0.000,C 180.000} C_DIS
LIN {X 2.500,Y 149.991,Z 49.000,A 180.000,B 0.000,C 180.000} C_DIS
LIN {X 2.506,Y 150.170,Z 49.000,A 180.000,B 0.000,C 180.000} C_DIS
LIN {X 2.506,Y 150.173,Z 49.000,A 180.000,B 0.000,C 180.000} C_DIS
LIN {X 2.524,Y 150.349,Z 49.000,A 180.000,B 0.000,C 180.000} C_DIS
LIN {X 2.556,Y 150.528,Z 49.000,A 180.000,B 0.000,C 180.000} C_DIS
LIN {X 2.602,Y 150.706,Z 49.000,A 180.000,B 0.000,C 180.000} C_DIS
LIN {X 2.662,Y 150.885,Z 49.000,A 180.000,B 0.000,C 180.000} C_DIS
LIN {X 2.685,Y 150.943,Z 49.000,A 180.000,B 0.000,C 180.000} C_DIS
LIN {X 2.738,Y 151.064,Z 49.000,A 180.000,B 0.000,C 180.000} C_DIS
LIN {X 2.831,Y 151.243,Z 49.000,A 180.000,B 0.000,C 180.000} C_DIS
LIN {X 2.864,Y 151.298,Z 49.000,A 180.000,B 0.000,C 180.000} C_DIS
LIN {X 2.943,Y 151.421,Z 49.000,A 180.000,B 0.000,C 180.000} C_DIS
LIN {X 3.042,Y 151.555,Z 49.000,A 180.000,B 0.000,C 180.000} C_DIS
LIN {X 3.079,Y 151.600,Z 49.000,A 180.000,B 0.000,C 180.000} C_DIS
LIN {X 3.221,Y 151.757,Z 49.000,A 180.000,B 0.000,C 180.000} C_DIS
LIN {X 3.243,Y 151.779,Z 49.000,A 180.000,B 0.000,C 180.000} C_DIS
LIN {X 3.400,Y 151.921,Z 49.000,A 180.000,B 0.000,C 180.000} C_DIS
LIN {X 3.445,Y 151.958,Z 49.000,A 180.000,B 0.000,C 180.000} C_DIS
LIN {X 3.579,Y 152.057,Z 49.000,A 180.000,B 0.000,C 180.000} C_DIS
LIN {X 3.702,Y 152.136,Z 49.000,A 180.000,B 0.000,C 180.000} C_DIS
LIN {X 3.757,Y 152.169,Z 49.000,A 180.000,B 0.000,C 180.000} C_DIS
LIN {X 3.936,Y 152.262,Z 49.000,A 180.000,B 0.000,C 180.000} C_DIS
LIN {X 4.057,Y 152.315,Z 49.000,A 180.000,B 0.000,C 180.000} C_DIS
LIN {X 4.115,Y 152.338,Z 49.000,A 180.000,B 0.000,C 180.000} C_DIS
LIN {X 4.294,Y 152.398,Z 49.000,A 180.000,B 0.000,C 180.000} C_DIS
LIN {X 4.472,Y 152.444,Z 49.000,A 180.000,B 0.000,C 180.000} C_DIS
LIN {X 4.651,Y 152.476,Z 49.000,A 180.000,B 0.000,C 180.000} C_DIS
LIN {X 4.827,Y 152.494,Z 49.000,A 180.000,B 0.000,C 180.000} C_DIS
LIN {X 4.830,Y 152.494,Z 49.000,A 180.000,B 0.000,C 180.000} C_DIS
LIN {X 5.009,Y 152.500,Z 49.000,A 180.000,B 0.000,C 180.000} C_DIS
LIN {X 149.991,Y 152.500,Z 49.000,A 180.000,B 0.000,C 180.000} C_DIS
LIN {X 150.170,Y 152.494,Z 49.000,A 180.000,B 0.000,C 180.000} C_DIS
LIN {X 150.173,Y 152.494,Z 49.000,A 180.000,B 0.000,C 180.000} C_DIS
LIN {X 150.349,Y 152.476,Z 49.000,A 180.000,B 0.000,C 180.000} C_DIS
LIN {X 150.528,Y 152.444,Z 49.000,A 180.000,B 0.000,C 180.000} C_DIS
LIN {X 150.706,Y 152.398,Z 49.000,A 180.000,B 0.000,C 180.000} C_DIS
LIN {X 150.885,Y 152.338,Z 49.000,A 180.000,B 0.000,C 180.000} C_DIS
LIN {X 150.943,Y 152.315,Z 49.000,A 180.000,B 0.000,C 180.000} C_DIS
LIN {X 151.064,Y 152.262,Z 49.000,A 180.000,B 0.000,C 180.000} C_DIS
LIN {X 151.243,Y 152.169,Z 49.000,A 180.000,B 0.000,C 180.000} C_DIS
LIN {X 151.298,Y 152.136,Z 49.000,A 180.000,B 0.000,C 180.000} C_DIS
LIN {X 151.421,Y 152.057,Z 49.000,A 180.000,B 0.000,C 180.000} C_DIS
LIN {X 151.555,Y 151.958,Z 49.000,A 180.000,B 0.000,C 180.000} C_DIS
LIN {X 151.600,Y 151.921,Z 49.000,A 180.000,B 0.000,C 180.000} C_DIS
LIN {X 151.757,Y 151.779,Z 49.000,A 180.000,B 0.000,C 180.000} C_DIS
LIN {X 151.779,Y 151.757,Z 49.000,A 180.000,B 0.000,C 180.000} C_DIS
LIN {X 151.921,Y 151.600,Z 49.000,A 180.000,B 0.000,C 180.000} C_DIS
LIN {X 151.958,Y 151.555,Z 49.000,A 180.000,B 0.000,C 180.000} C_DIS
LIN {X 152.057,Y 151.421,Z 49.000,A 180.000,B 0.000,C 180.000} C_DIS
LIN {X 152.136,Y 151.298,Z 49.000,A 180.000,B 0.000,C 180.000} C_DIS
LIN {X 152.169,Y 151.243,Z 49.000,A 180.000,B 0.000,C 180.000} C_DIS
LIN {X 152.262,Y 151.064,Z 49.000,A 180.000,B 0.000,C 180.000} C_DIS
LIN {X 152.315,Y 150.943,Z 49.000,A 180.000,B 0.000,C 180.000} C_DIS
LIN {X 152.338,Y 150.885,Z 49.000,A 180.000,B 0.000,C 180.000} C_DIS
LIN {X 152.398,Y 150.706,Z 49.000,A 180.000,B 0.000,C 180.000} C_DIS
LIN {X 152.444,Y 150.528,Z 49.000,A 180.000,B 0.000,C 180.000} C_DIS
LIN {X 152.476,Y 150.349,Z 49.000,A 180.000,B 0.000,C 180.000} C_DIS
LIN {X 152.494,Y 150.173,Z 49.000,A 180.000,B 0.000,C 180.000} C_DIS
LIN {X 152.494,Y 150.170,Z 49.000,A 180.000,B 0.000,C 180.000} C_DIS
LIN {X 152.500,Y 149.991,Z 49.000,A 180.000,B 0.000,C 180.000} C_DIS
LIN {X 152.500,Y 35.611,Z 49.000,A 180.000,B 0.000,C 180.000} C_DIS
LIN {X 152.500,Y 5.009,Z 49.000,A 180.000,B 0.000,C 180.000} C_DIS
LIN {X 152.494,Y 4.830,Z 49.000,A 180.000,B 0.000,C 180.000} C_DIS
LIN {X 152.494,Y 4.827,Z 49.000,A 180.000,B 0.000,C 180.000} C_DIS
LIN {X 152.476,Y 4.651,Z 49.000,A 180.000,B 0.000,C 180.000} C_DIS
LIN {X 152.444,Y 4.472,Z 49.000,A 180.000,B 0.000,C 180.000} C_DIS
LIN {X 152.398,Y 4.294,Z 49.000,A 180.000,B 0.000,C 180.000} C_DIS
LIN {X 152.338,Y 4.115,Z 49.000,A 180.000,B 0.000,C 180.000} C_DIS
LIN {X 152.315,Y 4.057,Z 49.000,A 180.000,B 0.000,C 180.000} C_DIS
LIN {X 152.262,Y 3.936,Z 49.000,A 180.000,B 0.000,C 180.000} C_DIS
LIN {X 152.169,Y 3.757,Z 49.000,A 180.000,B 0.000,C 180.000} C_DIS
LIN {X 152.136,Y 3.702,Z 49.000,A 180.000,B 0.000,C 180.000} C_DIS
LIN {X 152.057,Y 3.579,Z 49.000,A 180.000,B 0.000,C 180.000} C_DIS
LIN {X 151.958,Y 3.445,Z 49.000,A 180.000,B 0.000,C 180.000} C_DIS
LIN {X 151.921,Y 3.400,Z 49.000,A 180.000,B 0.000,C 180.000} C_DIS
LIN {X 151.779,Y 3.243,Z 49.000,A 180.000,B 0.000,C 180.000} C_DIS
LIN {X 151.757,Y 3.221,Z 49.000,A 180.000,B 0.000,C 180.000} C_DIS
LIN {X 151.600,Y 3.079,Z 49.000,A 180.000,B 0.000,C 180.000} C_DIS
LIN {X 151.555,Y 3.042,Z 49.000,A 180.000,B 0.000,C 180.000} C_DIS
LIN {X 151.421,Y 2.943,Z 49.000,A 180.000,B 0.000,C 180.000} C_DIS
LIN {X 151.298,Y 2.864,Z 49.000,A 180.000,B 0.000,C 180.000} C_DIS
LIN {X 151.243,Y 2.831,Z 49.000,A 180.000,B 0.000,C 180.000} C_DIS
LIN {X 151.064,Y 2.738,Z 49.000,A 180.000,B 0.000,C 180.000} C_DIS
LIN {X 150.943,Y 2.685,Z 49.000,A 180.000,B 0.000,C 180.000} C_DIS
LIN {X 150.885,Y 2.662,Z 49.000,A 180.000,B 0.000,C 180.000} C_DIS
LIN {X 150.706,Y 2.602,Z 49.000,A 180.000,B 0.000,C 180.000} C_DIS
LIN {X 150.528,Y 2.556,Z 49.000,A 180.000,B 0.000,C 180.000} C_DIS
LIN {X 150.349,Y 2.524,Z 49.000,A 180.000,B 0.000,C 180.000} C_DIS
LIN {X 150.173,Y 2.506,Z 49.000,A 180.000,B 0.000,C 180.000} C_DIS
LIN {X 150.170,Y 2.506,Z 49.000,A 180.000,B 0.000,C 180.000} C_DIS
LIN {X 149.991,Y 2.500,Z 49.000,A 180.000,B 0.000,C 180.000} C_DIS
LIN {X 147.452,Y 2.500,Z 49.000,A 180.000,B 0.000,C 180.000} C_DIS
; Link Move Starts
LIN {X 147.137,Y 2.500,Z 49.000,A 180.000,B 0.000,C 180.000} C_DIS
LIN {X 146.822,Y 2.500,Z 48.999,A 180.000,B 0.000,C 180.000} C_DIS
LIN {X 146.507,Y 2.500,Z 48.998,A 180.000,B 0.000,C 180.000} C_DIS
LIN {X 146.192,Y 2.500,Z 48.996,A 180.000,B 0.000,C 180.000} C_DIS
LIN {X 145.877,Y 2.500,Z 48.994,A 180.000,B 0.000,C 180.000} C_DIS
LIN {X 145.562,Y 2.500,Z 48.991,A 180.000,B 0.000,C 180.000} C_DIS
LIN {X 145.247,Y 2.500,Z 48.988,A 180.000,B 0.000,C 180.000} C_DIS
LIN {X 144.932,Y 2.500,Z 48.985,A 180.000,B 0.000,C 180.000} C_DIS
LIN {X 144.617,Y 2.500,Z 48.981,A 180.000,B 0.000,C 180.000} C_DIS
LIN {X 144.302,Y 2.500,Z 48.977,A 180.000,B 0.000,C 180.000} C_DIS
LIN {X 143.987,Y 2.500,Z 48.972,A 180.000,B 0.000,C 180.000} C_DIS
LIN {X 143.829,Y 2.500,Z 48.969,A 180.000,B 0.000,C 180.000} C_DIS
LIN {X 143.672,Y 2.500,Z 48.967,A 180.000,B 0.000,C 180.000} C_DIS
LIN {X 143.514,Y 2.500,Z 48.964,A 180.000,B 0.000,C 180.000} C_DIS
LIN {X 143.357,Y 2.500,Z 48.961,A 180.000,B 0.000,C 180.000} C_DIS
LIN {X 143.199,Y 2.500,Z 48.959,A 180.000,B 0.000,C 180.000} C_DIS
LIN {X 143.042,Y 2.500,Z 48.956,A 180.000,B 0.000,C 180.000} C_DIS
LIN {X 142.884,Y 2.500,Z 48.952,A 180.000,B 0.000,C 180.000} C_DIS
LIN {X 142.727,Y 2.500,Z 48.949,A 180.000,B 0.000,C 180.000} C_DIS
LIN {X 142.569,Y 2.500,Z 48.946,A 180.000,B 0.000,C 180.000} C_DIS
LIN {X 142.412,Y 2.500,Z 48.943,A 180.000,B 0.000,C 180.000} C_DIS
LIN {X 142.254,Y 2.500,Z 48.939,A 180.000,B 0.000,C 180.000} C_DIS
LIN {X 142.097,Y 2.500,Z 48.936,A 180.000,B 0.000,C 180.000} C_DIS
LIN {X 141.939,Y 2.500,Z 48.932,A 180.000,B 0.000,C 180.000} C_DIS
LIN {X 141.782,Y 2.500,Z 48.928,A 180.000,B 0.000,C 180.000} C_DIS
LIN {X 141.624,Y 2.500,Z 48.925,A 180.000,B 0.000,C 180.000} C_DIS
LIN {X 141.467,Y 2.500,Z 48.921,A 180.000,B 0.000,C 180.000} C_DIS
LIN {X 141.309,Y 2.500,Z 48.917,A 180.000,B 0.000,C 180.000} C_DIS
LIN {X 141.152,Y 2.500,Z 48.913,A 180.000,B 0.000,C 180.000} C_DIS
LIN {X 140.994,Y 2.500,Z 48.909,A 180.000,B 0.000,C 180.000} C_DIS
LIN {X 140.837,Y 2.500,Z 48.905,A 180.000,B 0.000,C 180.000} C_DIS
LIN {X 140.679,Y 2.500,Z 48.900,A 180.000,B 0.000,C 180.000} C_DIS
LIN {X 140.522,Y 2.500,Z 48.896,A 180.000,B 0.000,C 180.000} C_DIS
LIN {X 140.364,Y 2.500,Z 48.892,A 180.000,B 0.000,C 180.000} C_DIS
LIN {X 140.207,Y 2.500,Z 48.887,A 180.000,B 0.000,C 180.000} C_DIS
LIN {X 140.049,Y 2.500,Z 48.883,A 180.000,B 0.000,C 180.000} C_DIS
LIN {X 139.892,Y 2.500,Z 48.878,A 180.000,B 0.000,C 180.000} C_DIS
LIN {X 139.734,Y 2.500,Z 48.873,A 180.000,B 0.000,C 180.000} C_DIS
LIN {X 139.577,Y 2.500,Z 48.869,A 180.000,B 0.000,C 180.000} C_DIS
LIN {X 139.419,Y 2.500,Z 48.864,A 180.000,B 0.000,C 180.000} C_DIS
LIN {X 139.262,Y 2.500,Z 48.859,A 180.000,B 0.000,C 180.000} C_DIS
LIN {X 139.104,Y 2.500,Z 48.854,A 180.000,B 0.000,C 180.000} C_DIS
LIN {X 139.026,Y 2.500,Z 48.851,A 180.000,B 0.000,C 180.000} C_DIS
LIN {X 138.947,Y 2.500,Z 48.849,A 180.000,B 0.000,C 180.000} C_DIS
LIN {X 138.868,Y 2.500,Z 48.846,A 180.000,B 0.000,C 180.000} C_DIS
LIN {X 138.789,Y 2.500,Z 48.844,A 180.000,B 0.000,C 180.000} C_DIS
LIN {X 138.711,Y 2.500,Z 48.841,A 180.000,B 0.000,C 180.000} C_DIS
LIN {X 138.632,Y 2.500,Z 48.839,A 180.000,B 0.000,C 180.000} C_DIS
LIN {X 138.553,Y 2.500,Z 48.836,A 180.000,B 0.000,C 180.000} C_DIS
LIN {X 138.396,Y 2.500,Z 48.831,A 180.000,B 0.000,C 180.000} C_DIS
LIN {X 138.238,Y 2.500,Z 48.825,A 180.000,B 0.000,C 180.000} C_DIS
LIN {X 138.081,Y 2.500,Z 48.820,A 180.000,B 0.000,C 180.000} C_DIS
LIN {X 137.923,Y 2.500,Z 48.815,A 180.000,B 0.000,C 180.000} C_DIS
LIN {X 137.766,Y 2.500,Z 48.809,A 180.000,B 0.000,C 180.000} C_DIS
LIN {X 137.687,Y 2.500,Z 48.806,A 180.000,B 0.000,C 180.000} C_DIS
LIN {X 137.529,Y 2.500,Z 48.801,A 180.000,B 0.000,C 180.000} C_DIS
LIN {X 137.293,Y 2.500,Z 48.793,A 180.000,B 0.000,C 180.000} C_DIS
LIN {X 137.136,Y 2.500,Z 48.787,A 180.000,B 0.000,C 180.000} C_DIS
LIN {X 137.057,Y 2.500,Z 48.785,A 180.000,B 0.000,C 180.000} C_DIS
LIN {X 136.899,Y 2.500,Z 48.779,A 180.000,B 0.000,C 180.000} C_DIS
LIN {X 136.663,Y 2.500,Z 48.771,A 180.000,B 0.000,C 180.000} C_DIS
LIN {X 136.506,Y 2.500,Z 48.765,A 180.000,B 0.000,C 180.000} C_DIS
LIN {X 136.427,Y 2.500,Z 48.763,A 180.000,B 0.000,C 180.000} C_DIS
LIN {X 136.269,Y 2.500,Z 48.757,A 180.000,B 0.000,C 180.000} C_DIS
LIN {X 136.033,Y 2.500,Z 48.749,A 180.000,B 0.000,C 180.000} C_DIS
LIN {X 135.876,Y 2.500,Z 48.743,A 180.000,B 0.000,C 180.000} C_DIS
LIN {X 135.797,Y 2.500,Z 48.741,A 180.000,B 0.000,C 180.000} C_DIS
LIN {X 135.639,Y 2.500,Z 48.735,A 180.000,B 0.000,C 180.000} C_DIS
LIN {X 135.403,Y 2.500,Z 48.727,A 180.000,B 0.000,C 180.000} C_DIS
LIN {X 135.246,Y 2.500,Z 48.721,A 180.000,B 0.000,C 180.000} C_DIS
LIN {X 135.167,Y 2.500,Z 48.719,A 180.000,B 0.000,C 180.000} C_DIS
LIN {X 135.009,Y 2.500,Z 48.713,A 180.000,B 0.000,C 180.000} C_DIS
LIN {X 134.537,Y 2.500,Z 48.697,A 180.000,B 0.000,C 180.000} C_DIS
LIN {X 134.379,Y 2.500,Z 48.691,A 180.000,B 0.000,C 180.000} C_DIS
LIN {X 133.907,Y 2.500,Z 48.675,A 180.000,B 0.000,C 180.000} C_DIS
LIN {X 133.749,Y 2.500,Z 48.669,A 180.000,B 0.000,C 180.000} C_DIS
LIN {X 133.198,Y 2.500,Z 48.650,A 180.000,B 0.000,C 180.000} C_DIS
LIN {X 132.726,Y 2.500,Z 48.633,A 180.000,B 0.000,C 180.000} C_DIS
LIN {X 132.568,Y 2.500,Z 48.628,A 180.000,B 0.000,C 180.000} C_DIS
LIN {X 132.096,Y 2.500,Z 48.611,A 180.000,B 0.000,C 180.000} C_DIS
LIN {X 131.938,Y 2.500,Z 48.606,A 180.000,B 0.000,C 180.000} C_DIS
LIN {X 131.151,Y 2.500,Z 48.578,A 180.000,B 0.000,C 180.000} C_DIS
LIN {X 130.757,Y 2.500,Z 48.565,A 180.000,B 0.000,C 180.000} C_DIS
LIN {X 130.284,Y 2.500,Z 48.548,A 180.000,B 0.000,C 180.000} C_DIS
LIN {X 128.473,Y 2.500,Z 48.485,A 180.000,B 0.000,C 180.000} C_DIS
LIN {X 125.481,Y 2.500,Z 48.380,A 180.000,B 0.000,C 180.000} C_DIS
LIN {X 125.323,Y 2.500,Z 48.375,A 180.000,B 0.000,C 180.000} C_DIS
LIN {X 124.851,Y 2.500,Z 48.358,A 180.000,B 0.000,C 180.000} C_DIS
LIN {X 124.693,Y 2.500,Z 48.353,A 180.000,B 0.000,C 180.000} C_DIS
LIN {X 124.221,Y 2.500,Z 48.336,A 180.000,B 0.000,C 180.000} C_DIS
LIN {X 124.142,Y 2.500,Z 48.334,A 180.000,B 0.000,C 180.000} C_DIS
LIN {X 123.984,Y 2.500,Z 48.328,A 180.000,B 0.000,C 180.000} C_DIS
LIN {X 123.512,Y 2.500,Z 48.312,A 180.000,B 0.000,C 180.000} C_DIS
LIN {X 123.354,Y 2.500,Z 48.306,A 180.000,B 0.000,C 180.000} C_DIS
LIN {X 122.882,Y 2.500,Z 48.290,A 180.000,B 0.000,C 180.000} C_DIS
LIN {X 122.724,Y 2.500,Z 48.284,A 180.000,B 0.000,C 180.000} C_DIS
LIN {X 122.488,Y 2.500,Z 48.276,A 180.000,B 0.000,C 180.000} C_DIS
LIN {X 122.331,Y 2.500,Z 48.270,A 180.000,B 0.000,C 180.000} C_DIS
LIN {X 122.252,Y 2.500,Z 48.268,A 180.000,B 0.000,C 180.000} C_DIS
LIN {X 122.094,Y 2.500,Z 48.262,A 180.000,B 0.000,C 180.000} C_DIS
LIN {X 121.858,Y 2.500,Z 48.254,A 180.000,B 0.000,C 180.000} C_DIS
LIN {X 121.701,Y 2.500,Z 48.248,A 180.000,B 0.000,C 180.000} C_DIS
LIN {X 121.622,Y 2.500,Z 48.246,A 180.000,B 0.000,C 180.000} C_DIS
LIN {X 121.464,Y 2.500,Z 48.240,A 180.000,B 0.000,C 180.000} C_DIS
LIN {X 121.228,Y 2.500,Z 48.232,A 180.000,B 0.000,C 180.000} C_DIS
LIN {X 121.071,Y 2.500,Z 48.226,A 180.000,B 0.000,C 180.000} C_DIS
LIN {X 120.992,Y 2.500,Z 48.224,A 180.000,B 0.000,C 180.000} C_DIS
LIN {X 120.834,Y 2.500,Z 48.218,A 180.000,B 0.000,C 180.000} C_DIS
LIN {X 120.598,Y 2.500,Z 48.210,A 180.000,B 0.000,C 180.000} C_DIS
LIN {X 120.441,Y 2.500,Z 48.204,A 180.000,B 0.000,C 180.000} C_DIS
LIN {X 120.362,Y 2.500,Z 48.202,A 180.000,B 0.000,C 180.000} C_DIS
LIN {X 120.204,Y 2.500,Z 48.196,A 180.000,B 0.000,C 180.000} C_DIS
LIN {X 120.047,Y 2.500,Z 48.191,A 180.000,B 0.000,C 180.000} C_DIS
LIN {X 119.889,Y 2.500,Z 48.185,A 180.000,B 0.000,C 180.000} C_DIS
LIN {X 119.732,Y 2.500,Z 48.180,A 180.000,B 0.000,C 180.000} C_DIS
LIN {X 119.574,Y 2.500,Z 48.174,A 180.000,B 0.000,C 180.000} C_DIS
LIN {X 119.417,Y 2.500,Z 48.169,A 180.000,B 0.000,C 180.000} C_DIS
LIN {X 119.259,Y 2.500,Z 48.164,A 180.000,B 0.000,C 180.000} C_DIS
LIN {X 119.181,Y 2.500,Z 48.161,A 180.000,B 0.000,C 180.000} C_DIS
LIN {X 119.102,Y 2.500,Z 48.159,A 180.000,B 0.000,C 180.000} C_DIS
LIN {X 119.023,Y 2.500,Z 48.156,A 180.000,B 0.000,C 180.000} C_DIS
LIN {X 118.944,Y 2.500,Z 48.154,A 180.000,B 0.000,C 180.000} C_DIS
LIN {X 118.866,Y 2.500,Z 48.151,A 180.000,B 0.000,C 180.000} C_DIS
LIN {X 118.787,Y 2.500,Z 48.148,A 180.000,B 0.000,C 180.000} C_DIS
LIN {X 118.629,Y 2.500,Z 48.143,A 180.000,B 0.000,C 180.000} C_DIS
LIN {X 118.472,Y 2.500,Z 48.139,A 180.000,B 0.000,C 180.000} C_DIS
LIN {X 118.314,Y 2.500,Z 48.134,A 180.000,B 0.000,C 180.000} C_DIS
LIN {X 118.157,Y 2.500,Z 48.129,A 180.000,B 0.000,C 180.000} C_DIS
LIN {X 117.999,Y 2.500,Z 48.124,A 180.000,B 0.000,C 180.000} C_DIS
LIN {X 117.842,Y 2.500,Z 48.120,A 180.000,B 0.000,C 180.000} C_DIS
LIN {X 117.684,Y 2.500,Z 48.115,A 180.000,B 0.000,C 180.000} C_DIS
LIN {X 117.527,Y 2.500,Z 48.110,A 180.000,B 0.000,C 180.000} C_DIS
LIN {X 117.369,Y 2.500,Z 48.106,A 180.000,B 0.000,C 180.000} C_DIS
LIN {X 117.212,Y 2.500,Z 48.102,A 180.000,B 0.000,C 180.000} C_DIS
LIN {X 117.054,Y 2.500,Z 48.097,A 180.000,B 0.000,C 180.000} C_DIS
LIN {X 116.897,Y 2.500,Z 48.093,A 180.000,B 0.000,C 180.000} C_DIS
LIN {X 116.739,Y 2.500,Z 48.089,A 180.000,B 0.000,C 180.000} C_DIS
LIN {X 116.582,Y 2.500,Z 48.085,A 180.000,B 0.000,C 180.000} C_DIS
LIN {X 116.424,Y 2.500,Z 48.081,A 180.000,B 0.000,C 180.000} C_DIS
LIN {X 116.267,Y 2.500,Z 48.077,A 180.000,B 0.000,C 180.000} C_DIS
LIN {X 116.109,Y 2.500,Z 48.073,A 180.000,B 0.000,C 180.000} C_DIS
LIN {X 115.952,Y 2.500,Z 48.070,A 180.000,B 0.000,C 180.000} C_DIS
LIN {X 115.795,Y 2.500,Z 48.066,A 180.000,B 0.000,C 180.000} C_DIS
LIN {X 115.637,Y 2.500,Z 48.062,A 180.000,B 0.000,C 180.000} C_DIS
LIN {X 115.479,Y 2.500,Z 48.059,A 180.000,B 0.000,C 180.000} C_DIS
LIN {X 115.322,Y 2.500,Z 48.056,A 180.000,B 0.000,C 180.000} C_DIS
LIN {X 115.165,Y 2.500,Z 48.052,A 180.000,B 0.000,C 180.000} C_DIS
LIN {X 115.007,Y 2.500,Z 48.049,A 180.000,B 0.000,C 180.000} C_DIS
LIN {X 114.850,Y 2.500,Z 48.046,A 180.000,B 0.000,C 180.000} C_DIS
LIN {X 114.692,Y 2.500,Z 48.043,A 180.000,B 0.000,C 180.000} C_DIS
LIN {X 114.535,Y 2.500,Z 48.040,A 180.000,B 0.000,C 180.000} C_DIS
LIN {X 114.377,Y 2.500,Z 48.037,A 180.000,B 0.000,C 180.000} C_DIS
LIN {X 114.220,Y 2.500,Z 48.034,A 180.000,B 0.000,C 180.000} C_DIS
LIN {X 114.062,Y 2.500,Z 48.032,A 180.000,B 0.000,C 180.000} C_DIS
LIN {X 113.905,Y 2.500,Z 48.029,A 180.000,B 0.000,C 180.000} C_DIS
LIN {X 113.747,Y 2.500,Z 48.027,A 180.000,B 0.000,C 180.000} C_DIS
LIN {X 113.432,Y 2.500,Z 48.022,A 180.000,B 0.000,C 180.000} C_DIS
LIN {X 113.117,Y 2.500,Z 48.018,A 180.000,B 0.000,C 180.000} C_DIS
LIN {X 112.802,Y 2.500,Z 48.014,A 180.000,B 0.000,C 180.000} C_DIS
LIN {X 112.487,Y 2.500,Z 48.011,A 180.000,B 0.000,C 180.000} C_DIS
LIN {X 112.172,Y 2.500,Z 48.008,A 180.000,B 0.000,C 180.000} C_DIS
LIN {X 111.857,Y 2.500,Z 48.005,A 180.000,B 0.000,C 180.000} C_DIS
LIN {X 111.542,Y 2.500,Z 48.003,A 180.000,B 0.000,C 180.000} C_DIS
LIN {X 111.227,Y 2.500,Z 48.002,A 180.000,B 0.000,C 180.000} C_DIS
LIN {X 110.912,Y 2.500,Z 48.001,A 180.000,B 0.000,C 180.000} C_DIS
LIN {X 110.597,Y 2.500,Z 48.000,A 180.000,B 0.000,C 180.000} C_DIS
LIN {X 110.366,Y 2.500,Z 48.000,A 180.000,B 0.000,C 180.000} C_DIS
; Cutting Move Starts
LIN {X 5.009,Y 2.500,Z 48.000,A 180.000,B 0.000,C 180.000} C_DIS
LIN {X 4.830,Y 2.506,Z 48.000,A 180.000,B 0.000,C 180.000} C_DIS
LIN {X 4.827,Y 2.506,Z 48.000,A 180.000,B 0.000,C 180.000} C_DIS
LIN {X 4.651,Y 2.524,Z 48.000,A 180.000,B 0.000,C 180.000} C_DIS
LIN {X 4.472,Y 2.556,Z 48.000,A 180.000,B 0.000,C 180.000} C_DIS
LIN {X 4.294,Y 2.602,Z 48.000,A 180.000,B 0.000,C 180.000} C_DIS
LIN {X 4.115,Y 2.662,Z 48.000,A 180.000,B 0.000,C 180.000} C_DIS
LIN {X 4.057,Y 2.685,Z 48.000,A 180.000,B 0.000,C 180.000} C_DIS
LIN {X 3.936,Y 2.738,Z 48.000,A 180.000,B 0.000,C 180.000} C_DIS
LIN {X 3.757,Y 2.831,Z 48.000,A 180.000,B 0.000,C 180.000} C_DIS
LIN {X 3.702,Y 2.864,Z 48.000,A 180.000,B 0.000,C 180.000} C_DIS
LIN {X 3.579,Y 2.943,Z 48.000,A 180.000,B 0.000,C 180.000} C_DIS
LIN {X 3.445,Y 3.042,Z 48.000,A 180.000,B 0.000,C 180.000} C_DIS
LIN {X 3.400,Y 3.079,Z 48.000,A 180.000,B 0.000,C 180.000} C_DIS
LIN {X 3.243,Y 3.221,Z 48.000,A 180.000,B 0.000,C 180.000} C_DIS
LIN {X 3.221,Y 3.243,Z 48.000,A 180.000,B 0.000,C 180.000} C_DIS
LIN {X 3.079,Y 3.400,Z 48.000,A 180.000,B 0.000,C 180.000} C_DIS
LIN {X 3.042,Y 3.445,Z 48.000,A 180.000,B 0.000,C 180.000} C_DIS
LIN {X 2.943,Y 3.579,Z 48.000,A 180.000,B 0.000,C 180.000} C_DIS
LIN {X 2.864,Y 3.702,Z 48.000,A 180.000,B 0.000,C 180.000} C_DIS
LIN {X 2.831,Y 3.757,Z 48.000,A 180.000,B 0.000,C 180.000} C_DIS
LIN {X 2.738,Y 3.936,Z 48.000,A 180.000,B 0.000,C 180.000} C_DIS
LIN {X 2.685,Y 4.057,Z 48.000,A 180.000,B 0.000,C 180.000} C_DIS
LIN {X 2.662,Y 4.115,Z 48.000,A 180.000,B 0.000,C 180.000} C_DIS
LIN {X 2.602,Y 4.294,Z 48.000,A 180.000,B 0.000,C 180.000} C_DIS
LIN {X 2.556,Y 4.472,Z 48.000,A 180.000,B 0.000,C 180.000} C_DIS
LIN {X 2.524,Y 4.651,Z 48.000,A 180.000,B 0.000,C 180.000} C_DIS
LIN {X 2.506,Y 4.827,Z 48.000,A 180.000,B 0.000,C 180.000} C_DIS
LIN {X 2.506,Y 4.830,Z 48.000,A 180.000,B 0.000,C 180.000} C_DIS
LIN {X 2.500,Y 5.009,Z 48.000,A 180.000,B 0.000,C 180.000} C_DIS
LIN {X 2.500,Y 149.991,Z 48.000,A 180.000,B 0.000,C 180.000} C_DIS
LIN {X 2.506,Y 150.170,Z 48.000,A 180.000,B 0.000,C 180.000} C_DIS
LIN {X 2.506,Y 150.173,Z 48.000,A 180.000,B 0.000,C 180.000} C_DIS
LIN {X 2.524,Y 150.349,Z 48.000,A 180.000,B 0.000,C 180.000} C_DIS
LIN {X 2.556,Y 150.528,Z 48.000,A 180.000,B 0.000,C 180.000} C_DIS
LIN {X 2.602,Y 150.706,Z 48.000,A 180.000,B 0.000,C 180.000} C_DIS
LIN {X 2.662,Y 150.885,Z 48.000,A 180.000,B 0.000,C 180.000} C_DIS
LIN {X 2.685,Y 150.943,Z 48.000,A 180.000,B 0.000,C 180.000} C_DIS
LIN {X 2.738,Y 151.064,Z 48.000,A 180.000,B 0.000,C 180.000} C_DIS
LIN {X 2.831,Y 151.243,Z 48.000,A 180.000,B 0.000,C 180.000} C_DIS
LIN {X 2.864,Y 151.298,Z 48.000,A 180.000,B 0.000,C 180.000} C_DIS
LIN {X 2.943,Y 151.421,Z 48.000,A 180.000,B 0.000,C 180.000} C_DIS
LIN {X 3.042,Y 151.555,Z 48.000,A 180.000,B 0.000,C 180.000} C_DIS
LIN {X 3.079,Y 151.600,Z 48.000,A 180.000,B 0.000,C 180.000} C_DIS
LIN {X 3.221,Y 151.757,Z 48.000,A 180.000,B 0.000,C 180.000} C_DIS
LIN {X 3.243,Y 151.779,Z 48.000,A 180.000,B 0.000,C 180.000} C_DIS
LIN {X 3.400,Y 151.921,Z 48.000,A 180.000,B 0.000,C 180.000} C_DIS
LIN {X 3.445,Y 151.958,Z 48.000,A 180.000,B 0.000,C 180.000} C_DIS
LIN {X 3.579,Y 152.057,Z 48.000,A 180.000,B 0.000,C 180.000} C_DIS
LIN {X 3.702,Y 152.136,Z 48.000,A 180.000,B 0.000,C 180.000} C_DIS
LIN {X 3.757,Y 152.169,Z 48.000,A 180.000,B 0.000,C 180.000} C_DIS
LIN {X 3.936,Y 152.262,Z 48.000,A 180.000,B 0.000,C 180.000} C_DIS
LIN {X 4.057,Y 152.315,Z 48.000,A 180.000,B 0.000,C 180.000} C_DIS
LIN {X 4.115,Y 152.338,Z 48.000,A 180.000,B 0.000,C 180.000} C_DIS
LIN {X 4.294,Y 152.398,Z 48.000,A 180.000,B 0.000,C 180.000} C_DIS
LIN {X 4.472,Y 152.444,Z 48.000,A 180.000,B 0.000,C 180.000} C_DIS
LIN {X 4.651,Y 152.476,Z 48.000,A 180.000,B 0.000,C 180.000} C_DIS
LIN {X 4.827,Y 152.494,Z 48.000,A 180.000,B 0.000,C 180.000} C_DIS
LIN {X 4.830,Y 152.494,Z 48.000,A 180.000,B 0.000,C 180.000} C_DIS
LIN {X 5.009,Y 152.500,Z 48.000,A 180.000,B 0.000,C 180.000} C_DIS
LIN {X 149.991,Y 152.500,Z 48.000,A 180.000,B 0.000,C 180.000} C_DIS
LIN {X 150.170,Y 152.494,Z 48.000,A 180.000,B 0.000,C 180.000} C_DIS
LIN {X 150.173,Y 152.494,Z 48.000,A 180.000,B 0.000,C 180.000} C_DIS
LIN {X 150.349,Y 152.476,Z 48.000,A 180.000,B 0.000,C 180.000} C_DIS
LIN {X 150.528,Y 152.444,Z 48.000,A 180.000,B 0.000,C 180.000} C_DIS
LIN {X 150.706,Y 152.398,Z 48.000,A 180.000,B 0.000,C 180.000} C_DIS
LIN {X 150.885,Y 152.338,Z 48.000,A 180.000,B 0.000,C 180.000} C_DIS
LIN {X 150.943,Y 152.315,Z 48.000,A 180.000,B 0.000,C 180.000} C_DIS
LIN {X 151.064,Y 152.262,Z 48.000,A 180.000,B 0.000,C 180.000} C_DIS
LIN {X 151.243,Y 152.169,Z 48.000,A 180.000,B 0.000,C 180.000} C_DIS
LIN {X 151.298,Y 152.136,Z 48.000,A 180.000,B 0.000,C 180.000} C_DIS
LIN {X 151.421,Y 152.057,Z 48.000,A 180.000,B 0.000,C 180.000} C_DIS
LIN {X 151.555,Y 151.958,Z 48.000,A 180.000,B 0.000,C 180.000} C_DIS
LIN {X 151.600,Y 151.921,Z 48.000,A 180.000,B 0.000,C 180.000} C_DIS
LIN {X 151.757,Y 151.779,Z 48.000,A 180.000,B 0.000,C 180.000} C_DIS
LIN {X 151.779,Y 151.757,Z 48.000,A 180.000,B 0.000,C 180.000} C_DIS
LIN {X 151.921,Y 151.600,Z 48.000,A 180.000,B 0.000,C 180.000} C_DIS
LIN {X 151.958,Y 151.555,Z 48.000,A 180.000,B 0.000,C 180.000} C_DIS
LIN {X 152.057,Y 151.421,Z 48.000,A 180.000,B 0.000,C 180.000} C_DIS
LIN {X 152.136,Y 151.298,Z 48.000,A 180.000,B 0.000,C 180.000} C_DIS
LIN {X 152.169,Y 151.243,Z 48.000,A 180.000,B 0.000,C 180.000} C_DIS
LIN {X 152.262,Y 151.064,Z 48.000,A 180.000,B 0.000,C 180.000} C_DIS
LIN {X 152.315,Y 150.943,Z 48.000,A 180.000,B 0.000,C 180.000} C_DIS
LIN {X 152.338,Y 150.885,Z 48.000,A 180.000,B 0.000,C 180.000} C_DIS
LIN {X 152.398,Y 150.706,Z 48.000,A 180.000,B 0.000,C 180.000} C_DIS
LIN {X 152.444,Y 150.528,Z 48.000,A 180.000,B 0.000,C 180.000} C_DIS
LIN {X 152.476,Y 150.349,Z 48.000,A 180.000,B 0.000,C 180.000} C_DIS
LIN {X 152.494,Y 150.173,Z 48.000,A 180.000,B 0.000,C 180.000} C_DIS
LIN {X 152.494,Y 150.170,Z 48.000,A 180.000,B 0.000,C 180.000} C_DIS
LIN {X 152.500,Y 149.991,Z 48.000,A 180.000,B 0.000,C 180.000} C_DIS
LIN {X 152.500,Y 5.009,Z 48.000,A 180.000,B 0.000,C 180.000} C_DIS
LIN {X 152.494,Y 4.830,Z 48.000,A 180.000,B 0.000,C 180.000} C_DIS
LIN {X 152.494,Y 4.827,Z 48.000,A 180.000,B 0.000,C 180.000} C_DIS
LIN {X 152.476,Y 4.651,Z 48.000,A 180.000,B 0.000,C 180.000} C_DIS
LIN {X 152.444,Y 4.472,Z 48.000,A 180.000,B 0.000,C 180.000} C_DIS
LIN {X 152.398,Y 4.294,Z 48.000,A 180.000,B 0.000,C 180.000} C_DIS
LIN {X 152.338,Y 4.115,Z 48.000,A 180.000,B 0.000,C 180.000} C_DIS
LIN {X 152.315,Y 4.057,Z 48.000,A 180.000,B 0.000,C 180.000} C_DIS
LIN {X 152.262,Y 3.936,Z 48.000,A 180.000,B 0.000,C 180.000} C_DIS
LIN {X 152.169,Y 3.757,Z 48.000,A 180.000,B 0.000,C 180.000} C_DIS
LIN {X 152.136,Y 3.702,Z 48.000,A 180.000,B 0.000,C 180.000} C_DIS
LIN {X 152.057,Y 3.579,Z 48.000,A 180.000,B 0.000,C 180.000} C_DIS
LIN {X 151.958,Y 3.445,Z 48.000,A 180.000,B 0.000,C 180.000} C_DIS
LIN {X 151.921,Y 3.400,Z 48.000,A 180.000,B 0.000,C 180.000} C_DIS
LIN {X 151.779,Y 3.243,Z 48.000,A 180.000,B 0.000,C 180.000} C_DIS
LIN {X 151.757,Y 3.221,Z 48.000,A 180.000,B 0.000,C 180.000} C_DIS
LIN {X 151.600,Y 3.079,Z 48.000,A 180.000,B 0.000,C 180.000} C_DIS
LIN {X 151.555,Y 3.042,Z 48.000,A 180.000,B 0.000,C 180.000} C_DIS
LIN {X 151.421,Y 2.943,Z 48.000,A 180.000,B 0.000,C 180.000} C_DIS
LIN {X 151.298,Y 2.864,Z 48.000,A 180.000,B 0.000,C 180.000} C_DIS
LIN {X 151.243,Y 2.831,Z 48.000,A 180.000,B 0.000,C 180.000} C_DIS
LIN {X 151.064,Y 2.738,Z 48.000,A 180.000,B 0.000,C 180.000} C_DIS
LIN {X 150.943,Y 2.685,Z 48.000,A 180.000,B 0.000,C 180.000} C_DIS
LIN {X 150.885,Y 2.662,Z 48.000,A 180.000,B 0.000,C 180.000} C_DIS
LIN {X 150.706,Y 2.602,Z 48.000,A 180.000,B 0.000,C 180.000} C_DIS
LIN {X 150.528,Y 2.556,Z 48.000,A 180.000,B 0.000,C 180.000} C_DIS
LIN {X 150.349,Y 2.524,Z 48.000,A 180.000,B 0.000,C 180.000} C_DIS
LIN {X 150.173,Y 2.506,Z 48.000,A 180.000,B 0.000,C 180.000} C_DIS
LIN {X 150.170,Y 2.506,Z 48.000,A 180.000,B 0.000,C 180.000} C_DIS
LIN {X 149.991,Y 2.500,Z 48.000,A 180.000,B 0.000,C 180.000} C_DIS
LIN {X 110.366,Y 2.500,Z 48.000,A 180.000,B 0.000,C 180.000} C_DIS
; Link Move Starts
LIN {X 110.051,Y 2.500,Z 48.000,A 180.000,B 0.000,C 180.000} C_DIS
LIN {X 109.736,Y 2.500,Z 47.999,A 180.000,B 0.000,C 180.000} C_DIS
LIN {X 109.421,Y 2.500,Z 47.998,A 180.000,B 0.000,C 180.000} C_DIS
LIN {X 109.106,Y 2.500,Z 47.996,A 180.000,B 0.000,C 180.000} C_DIS
LIN {X 108.791,Y 2.500,Z 47.994,A 180.000,B 0.000,C 180.000} C_DIS
LIN {X 108.476,Y 2.500,Z 47.991,A 180.000,B 0.000,C 180.000} C_DIS
LIN {X 108.161,Y 2.500,Z 47.988,A 180.000,B 0.000,C 180.000} C_DIS
LIN {X 107.846,Y 2.500,Z 47.985,A 180.000,B 0.000,C 180.000} C_DIS
LIN {X 107.531,Y 2.500,Z 47.981,A 180.000,B 0.000,C 180.000} C_DIS
LIN {X 107.216,Y 2.500,Z 47.977,A 180.000,B 0.000,C 180.000} C_DIS
LIN {X 106.901,Y 2.500,Z 47.972,A 180.000,B 0.000,C 180.000} C_DIS
LIN {X 106.744,Y 2.500,Z 47.969,A 180.000,B 0.000,C 180.000} C_DIS
LIN {X 106.586,Y 2.500,Z 47.967,A 180.000,B 0.000,C 180.000} C_DIS
LIN {X 106.429,Y 2.500,Z 47.964,A 180.000,B 0.000,C 180.000} C_DIS
LIN {X 106.271,Y 2.500,Z 47.961,A 180.000,B 0.000,C 180.000} C_DIS
LIN {X 106.114,Y 2.500,Z 47.959,A 180.000,B 0.000,C 180.000} C_DIS
LIN {X 105.956,Y 2.500,Z 47.956,A 180.000,B 0.000,C 180.000} C_DIS
LIN {X 105.799,Y 2.500,Z 47.952,A 180.000,B 0.000,C 180.000} C_DIS
LIN {X 105.641,Y 2.500,Z 47.949,A 180.000,B 0.000,C 180.000} C_DIS
LIN {X 105.484,Y 2.500,Z 47.946,A 180.000,B 0.000,C 180.000} C_DIS
LIN {X 105.326,Y 2.500,Z 47.943,A 180.000,B 0.000,C 180.000} C_DIS
LIN {X 105.169,Y 2.500,Z 47.939,A 180.000,B 0.000,C 180.000} C_DIS
LIN {X 105.011,Y 2.500,Z 47.936,A 180.000,B 0.000,C 180.000} C_DIS
LIN {X 104.854,Y 2.500,Z 47.932,A 180.000,B 0.000,C 180.000} C_DIS
LIN {X 104.696,Y 2.500,Z 47.928,A 180.000,B 0.000,C 180.000} C_DIS
LIN {X 104.539,Y 2.500,Z 47.925,A 180.000,B 0.000,C 180.000} C_DIS
LIN {X 104.381,Y 2.500,Z 47.921,A 180.000,B 0.000,C 180.000} C_DIS
LIN {X 104.224,Y 2.500,Z 47.917,A 180.000,B 0.000,C 180.000} C_DIS
LIN {X 104.066,Y 2.500,Z 47.913,A 180.000,B 0.000,C 180.000} C_DIS
LIN {X 103.909,Y 2.500,Z 47.909,A 180.000,B 0.000,C 180.000} C_DIS
LIN {X 103.751,Y 2.500,Z 47.905,A 180.000,B 0.000,C 180.000} C_DIS
LIN {X 103.594,Y 2.500,Z 47.900,A 180.000,B 0.000,C 180.000} C_DIS
LIN {X 103.436,Y 2.500,Z 47.896,A 180.000,B 0.000,C 180.000} C_DIS
LIN {X 103.279,Y 2.500,Z 47.892,A 180.000,B 0.000,C 180.000} C_DIS
LIN {X 103.121,Y 2.500,Z 47.887,A 180.000,B 0.000,C 180.000} C_DIS
LIN {X 102.964,Y 2.500,Z 47.883,A 180.000,B 0.000,C 180.000} C_DIS
LIN {X 102.806,Y 2.500,Z 47.878,A 180.000,B 0.000,C 180.000} C_DIS
LIN {X 102.649,Y 2.500,Z 47.873,A 180.000,B 0.000,C 180.000} C_DIS
LIN {X 102.491,Y 2.500,Z 47.869,A 180.000,B 0.000,C 180.000} C_DIS
LIN {X 102.334,Y 2.500,Z 47.864,A 180.000,B 0.000,C 180.000} C_DIS
LIN {X 102.176,Y 2.500,Z 47.859,A 180.000,B 0.000,C 180.000} C_DIS
LIN {X 102.019,Y 2.500,Z 47.854,A 180.000,B 0.000,C 180.000} C_DIS
LIN {X 101.940,Y 2.500,Z 47.851,A 180.000,B 0.000,C 180.000} C_DIS
LIN {X 101.861,Y 2.500,Z 47.849,A 180.000,B 0.000,C 180.000} C_DIS
LIN {X 101.782,Y 2.500,Z 47.846,A 180.000,B 0.000,C 180.000} C_DIS
LIN {X 101.704,Y 2.500,Z 47.844,A 180.000,B 0.000,C 180.000} C_DIS
LIN {X 101.625,Y 2.500,Z 47.841,A 180.000,B 0.000,C 180.000} C_DIS
LIN {X 101.546,Y 2.500,Z 47.839,A 180.000,B 0.000,C 180.000} C_DIS
LIN {X 101.467,Y 2.500,Z 47.836,A 180.000,B 0.000,C 180.000} C_DIS
LIN {X 101.310,Y 2.500,Z 47.831,A 180.000,B 0.000,C 180.000} C_DIS
LIN {X 101.152,Y 2.500,Z 47.825,A 180.000,B 0.000,C 180.000} C_DIS
LIN {X 100.995,Y 2.500,Z 47.820,A 180.000,B 0.000,C 180.000} C_DIS
LIN {X 100.837,Y 2.500,Z 47.815,A 180.000,B 0.000,C 180.000} C_DIS
LIN {X 100.680,Y 2.500,Z 47.809,A 180.000,B 0.000,C 180.000} C_DIS
LIN {X 100.601,Y 2.500,Z 47.806,A 180.000,B 0.000,C 180.000} C_DIS
LIN {X 100.444,Y 2.500,Z 47.801,A 180.000,B 0.000,C 180.000} C_DIS
LIN {X 100.207,Y 2.500,Z 47.793,A 180.000,B 0.000,C 180.000} C_DIS
LIN {X 100.050,Y 2.500,Z 47.787,A 180.000,B 0.000,C 180.000} C_DIS
LIN {X 99.971,Y 2.500,Z 47.785,A 180.000,B 0.000,C 180.000} C_DIS
LIN {X 99.814,Y 2.500,Z 47.779,A 180.000,B 0.000,C 180.000} C_DIS
LIN {X 99.577,Y 2.500,Z 47.771,A 180.000,B 0.000,C 180.000} C_DIS
LIN {X 99.420,Y 2.500,Z 47.765,A 180.000,B 0.000,C 180.000} C_DIS
LIN {X 99.341,Y 2.500,Z 47.763,A 180.000,B 0.000,C 180.000} C_DIS
LIN {X 99.184,Y 2.500,Z 47.757,A 180.000,B 0.000,C 180.000} C_DIS
LIN {X 98.947,Y 2.500,Z 47.749,A 180.000,B 0.000,C 180.000} C_DIS
LIN {X 98.790,Y 2.500,Z 47.743,A 180.000,B 0.000,C 180.000} C_DIS
LIN {X 98.711,Y 2.500,Z 47.741,A 180.000,B 0.000,C 180.000} C_DIS
LIN {X 98.554,Y 2.500,Z 47.735,A 180.000,B 0.000,C 180.000} C_DIS
LIN {X 98.317,Y 2.500,Z 47.727,A 180.000,B 0.000,C 180.000} C_DIS
LIN {X 98.160,Y 2.500,Z 47.721,A 180.000,B 0.000,C 180.000} C_DIS
LIN {X 98.081,Y 2.500,Z 47.719,A 180.000,B 0.000,C 180.000} C_DIS
LIN {X 97.924,Y 2.500,Z 47.713,A 180.000,B 0.000,C 180.000} C_DIS
LIN {X 97.451,Y 2.500,Z 47.697,A 180.000,B 0.000,C 180.000} C_DIS
LIN {X 97.294,Y 2.500,Z 47.691,A 180.000,B 0.000,C 180.000} C_DIS
LIN {X 96.821,Y 2.500,Z 47.675,A 180.000,B 0.000,C 180.000} C_DIS
LIN {X 96.664,Y 2.500,Z 47.669,A 180.000,B 0.000,C 180.000} C_DIS
LIN {X 96.112,Y 2.500,Z 47.650,A 180.000,B 0.000,C 180.000} C_DIS
LIN {X 95.640,Y 2.500,Z 47.633,A 180.000,B 0.000,C 180.000} C_DIS
LIN {X 95.482,Y 2.500,Z 47.628,A 180.000,B 0.000,C 180.000} C_DIS
LIN {X 95.010,Y 2.500,Z 47.611,A 180.000,B 0.000,C 180.000} C_DIS
LIN {X 94.852,Y 2.500,Z 47.606,A 180.000,B 0.000,C 180.000} C_DIS
LIN {X 94.065,Y 2.500,Z 47.578,A 180.000,B 0.000,C 180.000} C_DIS
LIN {X 93.671,Y 2.500,Z 47.565,A 180.000,B 0.000,C 180.000} C_DIS
LIN {X 93.199,Y 2.500,Z 47.548,A 180.000,B 0.000,C 180.000} C_DIS
LIN {X 91.387,Y 2.500,Z 47.485,A 180.000,B 0.000,C 180.000} C_DIS
LIN {X 88.395,Y 2.500,Z 47.380,A 180.000,B 0.000,C 180.000} C_DIS
LIN {X 88.237,Y 2.500,Z 47.375,A 180.000,B 0.000,C 180.000} C_DIS
LIN {X 87.765,Y 2.500,Z 47.358,A 180.000,B 0.000,C 180.000} C_DIS
LIN {X 87.607,Y 2.500,Z 47.353,A 180.000,B 0.000,C 180.000} C_DIS
LIN {X 87.135,Y 2.500,Z 47.336,A 180.000,B 0.000,C 180.000} C_DIS
LIN {X 87.056,Y 2.500,Z 47.334,A 180.000,B 0.000,C 180.000} C_DIS
LIN {X 86.899,Y 2.500,Z 47.328,A 180.000,B 0.000,C 180.000} C_DIS
LIN {X 86.426,Y 2.500,Z 47.312,A 180.000,B 0.000,C 180.000} C_DIS
LIN {X 86.269,Y 2.500,Z 47.306,A 180.000,B 0.000,C 180.000} C_DIS
LIN {X 85.796,Y 2.500,Z 47.290,A 180.000,B 0.000,C 180.000} C_DIS
LIN {X 85.639,Y 2.500,Z 47.284,A 180.000,B 0.000,C 180.000} C_DIS
LIN {X 85.402,Y 2.500,Z 47.276,A 180.000,B 0.000,C 180.000} C_DIS
LIN {X 85.245,Y 2.500,Z 47.270,A 180.000,B 0.000,C 180.000} C_DIS
LIN {X 85.166,Y 2.500,Z 47.268,A 180.000,B 0.000,C 180.000} C_DIS
